C05477=1230.678,265.169,-62.603,-176.696,6.427,148.193
C05478=1230.673,265.417,-62.630,-176.693,6.429,148.193
C05479=1230.669,265.666,-62.657,-176.691,6.431,148.193
C05480=1230.665,265.914,-62.685,-176.689,6.433,148.193
C05481=1230.660,266.163,-62.713,-176.686,6.435,148.192
C05482=1230.656,266.411,-62.740,-176.684,6.437,148.192
C05483=1230.651,266.659,-62.767,-176.681,6.439,148.192
C05484=1230.647,266.908,-62.795,-176.679,6.441,148.192
C05485=1230.642,267.157,-62.822,-176.677,6.443,148.191
C05486=1230.638,267.405,-62.850,-176.674,6.445,148.191
C05487=1230.633,267.653,-62.877,-176.672,6.447,148.191
C05488=1230.629,267.903,-62.904,-176.669,6.449,148.191
C05489=1230.625,268.150,-62.932,-176.667,6.452,148.191
C05490=1230.620,268.399,-62.959,-176.664,6.454,148.190
C05491=1230.616,268.647,-62.987,-176.661,6.456,148.190
C05492=1230.612,268.896,-63.014,-176.659,6.458,148.190
C05493=1230.607,269.144,-63.041,-176.657,6.460,148.190
C05494=1230.603,269.392,-63.069,-176.655,6.462,148.190
C05495=1230.598,269.641,-63.096,-176.652,6.464,148.189
C05496=1230.595,269.889,-63.124,-176.649,6.466,148.189
C05497=1230.590,270.138,-63.151,-176.647,6.468,148.189
C05498=1230.585,270.386,-63.180,-176.645,6.470,148.189
C05499=1230.581,270.635,-63.207,-176.642,6.473,148.189
C05500=1230.576,270.883,-63.235,-176.639,6.475,148.188
C05501=1230.572,271.132,-63.262,-176.637,6.477,148.188
C05502=1230.568,271.380,-63.290,-176.635,6.479,148.188
C05503=1230.563,271.629,-63.317,-176.632,6.481,148.188
C05504=1230.559,271.877,-63.345,-176.630,6.483,148.188
C05505=1230.555,272.126,-63.374,-176.627,6.485,148.187
C05506=1230.550,272.374,-63.401,-176.625,6.487,148.187
C05507=1230.546,272.622,-63.428,-176.623,6.489,148.187
C05508=1230.541,272.871,-63.456,-176.620,6.492,148.187
C05509=1230.537,273.119,-63.484,-176.617,6.494,148.187
C05510=1230.533,273.367,-63.511,-176.615,6.496,148.187
C05511=1230.528,273.616,-63.539,-176.613,6.498,148.186
C05512=1230.524,273.864,-63.567,-176.610,6.500,148.186
C05513=1230.519,274.112,-63.595,-176.608,6.502,148.186
C05514=1230.515,274.361,-63.622,-176.605,6.504,148.186
C05515=1230.511,274.609,-63.650,-176.603,6.507,148.186
C05516=1230.506,274.858,-63.679,-176.600,6.509,148.185
C05517=1230.502,275.107,-63.706,-176.598,6.512,148.185
C05518=1230.497,275.354,-63.734,-176.595,6.513,148.185
C05519=1230.494,275.603,-63.762,-176.593,6.516,148.185
C05520=1230.489,275.851,-63.790,-176.591,6.518,148.185
C05521=1230.484,276.100,-63.818,-176.589,6.520,148.185
C05522=1230.480,276.348,-63.846,-176.586,6.522,148.184
C05523=1230.475,276.596,-63.874,-176.584,6.524,148.184
C05524=1230.471,276.845,-63.902,-176.581,6.527,148.184
C05525=1230.467,277.093,-63.929,-176.579,6.529,148.184
C05526=1230.463,277.342,-63.957,-176.576,6.531,148.184
C05527=1230.458,277.590,-63.986,-176.574,6.533,148.184
C05528=1230.454,277.839,-64.014,-176.571,6.535,148.183
C05529=1230.450,278.087,-64.042,-176.569,6.537,148.183
C05530=1230.445,278.335,-64.070,-176.567,6.539,148.183
C05531=1230.441,278.584,-64.097,-176.564,6.542,148.183
C05532=1230.436,278.832,-64.125,-176.561,6.544,148.183
C05533=1230.432,279.081,-64.154,-176.559,6.546,148.183
C05534=1230.427,279.329,-64.182,-176.557,6.548,148.182
C05535=1230.423,279.578,-64.210,-176.555,6.550,148.182
C05536=1230.419,279.825,-64.238,-176.552,6.552,148.182
C05537=1230.415,280.074,-64.266,-176.549,6.555,148.182
C05538=1230.410,280.322,-64.295,-176.547,6.557,148.182
C05539=1230.406,280.571,-64.323,-176.545,6.559,148.182
C05540=1230.401,280.819,-64.351,-176.543,6.562,148.181
C05541=1230.397,281.068,-64.379,-176.540,6.563,148.181
C05542=1230.393,281.315,-64.407,-176.538,6.566,148.181
C05543=1230.388,281.564,-64.436,-176.535,6.568,148.181
C05544=1230.384,281.812,-64.464,-176.533,6.571,148.181
C05545=1230.379,282.061,-64.492,-176.530,6.572,148.181
C05546=1230.375,282.309,-64.520,-176.528,6.575,148.180
C05547=1230.371,282.558,-64.549,-176.526,6.577,148.180
C05548=1230.366,282.806,-64.577,-176.523,6.579,148.180
C05549=1230.362,283.055,-64.605,-176.520,6.582,148.180
C05550=1230.357,283.303,-64.633,-176.518,6.584,148.180
C05551=1230.353,283.551,-64.662,-176.516,6.586,148.180
C05552=1230.349,283.799,-64.690,-176.513,6.588,148.179
C05553=1230.344,284.048,-64.718,-176.511,6.590,148.179
C05554=1230.340,284.297,-64.747,-176.509,6.592,148.179
C05555=1230.336,284.544,-64.776,-176.506,6.595,148.179
C05556=1230.332,284.793,-64.804,-176.504,6.597,148.179
C05557=1230.327,285.041,-64.832,-176.501,6.599,148.179
C05558=1230.323,285.290,-64.860,-176.499,6.601,148.179
C05559=1230.318,285.538,-64.889,-176.497,6.604,148.179
C05560=1230.314,285.786,-64.917,-176.494,6.606,148.178
C05561=1230.310,286.035,-64.946,-176.492,6.609,148.178
C05562=1230.305,286.283,-64.975,-176.490,6.611,148.178
C05563=1230.301,286.531,-65.003,-176.487,6.613,148.178
C05564=1230.296,286.780,-65.031,-176.485,6.615,148.178
C05565=1230.293,287.028,-65.060,-176.482,6.618,148.178
C05566=1230.288,287.276,-65.089,-176.480,6.620,148.178
C05567=1230.283,287.525,-65.117,-176.477,6.622,148.178
C05568=1230.279,287.773,-65.145,-176.475,6.624,148.177
C05569=1230.274,288.021,-65.174,-176.473,6.626,148.177
C05570=1230.271,288.269,-65.203,-176.470,6.629,148.177
C05571=1230.266,288.518,-65.231,-176.468,6.631,148.177
C05572=1230.261,288.766,-65.260,-176.465,6.633,148.177
C05573=1230.258,289.014,-65.288,-176.463,6.636,148.177
C05574=1230.253,289.289,-65.320,-176.460,6.638,148.177
C05575=1230.247,289.562,-65.351,-176.458,6.641,148.176
C05576=1230.243,289.836,-65.384,-176.455,6.643,148.176
C05577=1230.238,290.111,-65.415,-176.453,6.646,148.176
C05578=1230.234,290.359,-65.444,-176.450,6.647,148.176
C05579=1230.230,290.607,-65.473,-176.448,6.651,148.176
C05580=1230.225,290.856,-65.501,-176.445,6.653,148.176
C05581=1230.221,291.104,-65.530,-176.443,6.655,148.176
C05582=1230.216,291.352,-65.559,-176.441,6.657,148.175
C05583=1230.212,291.601,-65.587,-176.438,6.660,148.175
C05584=1230.208,291.849,-65.617,-176.436,6.662,148.175
C05585=1230.203,292.097,-65.645,-176.433,6.664,148.175
C05586=1230.199,292.345,-65.674,-176.431,6.666,148.175
C05587=1230.195,292.594,-65.703,-176.429,6.668,148.175
C05588=1230.191,292.842,-65.732,-176.426,6.671,148.175
C05589=1230.186,293.090,-65.761,-176.424,6.673,148.175
C05590=1230.181,293.339,-65.790,-176.422,6.676,148.175
C05591=1230.178,293.587,-65.818,-176.420,6.678,148.175
C05592=1230.173,293.835,-65.847,-176.417,6.681,148.174
C05593=1230.168,294.084,-65.876,-176.415,6.683,148.174
C05594=1230.164,294.332,-65.905,-176.412,6.685,148.174
C05595=1230.160,294.580,-65.935,-176.410,6.687,148.174
C05596=1230.156,294.828,-65.963,-176.408,6.689,148.174
C05597=1230.152,295.076,-65.992,-176.405,6.692,148.174
C05598=1230.147,295.325,-66.021,-176.403,6.694,148.174
C05599=1230.143,295.573,-66.050,-176.401,6.697,148.174
C05600=1230.138,295.821,-66.079,-176.398,6.699,148.173
C05601=1230.134,296.070,-66.108,-176.396,6.702,148.173
C05602=1230.130,296.318,-66.137,-176.393,6.704,148.173
C05603=1230.126,296.566,-66.166,-176.391,6.706,148.173
C05604=1230.122,296.815,-66.195,-176.389,6.708,148.173
C05605=1230.117,297.063,-66.224,-176.386,6.711,148.173
C05606=1230.113,297.311,-66.254,-176.384,6.713,148.173
C05607=1230.108,297.559,-66.283,-176.382,6.715,148.173
C05608=1230.104,297.808,-66.312,-176.380,6.718,148.173
C05609=1230.100,298.056,-66.341,-176.377,6.720,148.173
C05610=1230.095,298.304,-66.370,-176.375,6.723,148.173
C05611=1230.091,298.552,-66.400,-176.372,6.725,148.173
C05612=1230.086,298.801,-66.429,-176.370,6.727,148.172
C05613=1230.082,299.049,-66.458,-176.368,6.730,148.172
C05614=1230.079,299.297,-66.487,-176.365,6.732,148.172
C05615=1230.074,299.545,-66.516,-176.363,6.734,148.172
C05616=1230.070,299.793,-66.546,-176.361,6.737,148.172
C05617=1230.065,300.041,-66.575,-176.358,6.740,148.172
C05618=1230.061,300.290,-66.604,-176.356,6.742,148.172
C05619=1230.057,300.538,-66.633,-176.354,6.744,148.172
C05620=1230.053,300.787,-66.663,-176.351,6.746,148.172
C05621=1230.048,301.034,-66.692,-176.349,6.749,148.172
C05622=1230.044,301.283,-66.721,-176.347,6.751,148.172
C05623=1230.039,301.531,-66.751,-176.345,6.753,148.172
C05624=1230.035,301.779,-66.781,-176.342,6.756,148.172
C05625=1230.030,302.028,-66.810,-176.340,6.759,148.172
C05626=1230.026,302.276,-66.840,-176.338,6.761,148.171
C05627=1230.022,302.524,-66.869,-176.336,6.763,148.171
C05628=1230.018,302.773,-66.898,-176.333,6.765,148.171
C05629=1230.013,303.021,-66.927,-176.330,6.768,148.171
C05630=1230.009,303.269,-66.956,-176.328,6.770,148.171
C05631=1230.004,303.517,-66.986,-176.326,6.773,148.171
C05632=1230.000,303.765,-67.015,-176.324,6.775,148.171
C05633=1229.996,304.014,-67.045,-176.321,6.778,148.171
C05634=1229.992,304.262,-67.074,-176.319,6.780,148.171
C05635=1229.988,304.510,-67.104,-176.317,6.782,148.171
C05636=1229.983,304.758,-67.134,-176.315,6.785,148.171
C05637=1229.979,305.007,-67.164,-176.312,6.788,148.171
C05638=1229.975,305.255,-67.193,-176.310,6.789,148.171
C05639=1229.970,305.502,-67.222,-176.308,6.792,148.170
C05640=1229.966,305.751,-67.252,-176.306,6.794,148.170
C05641=1229.962,305.999,-67.281,-176.303,6.797,148.170
C05642=1229.957,306.247,-67.311,-176.301,6.799,148.170
C05643=1229.952,306.496,-67.341,-176.299,6.801,148.170
C05644=1229.948,306.744,-67.370,-176.296,6.805,148.170
C05645=1229.944,306.992,-67.400,-176.294,6.807,148.170
C05646=1229.940,307.240,-67.430,-176.292,6.809,148.170
C05647=1229.936,307.488,-67.459,-176.290,6.811,148.170
C05648=1229.931,307.737,-67.489,-176.287,6.814,148.170
C05649=1229.927,307.985,-67.519,-176.285,6.816,148.170
C05650=1229.923,308.233,-67.548,-176.283,6.819,148.170
C05651=1229.919,308.481,-67.578,-176.280,6.822,148.170
C05652=1229.914,308.730,-67.608,-176.278,6.824,148.170
C05653=1229.910,308.978,-67.638,-176.276,6.826,148.170
C05654=1229.906,309.226,-67.667,-176.274,6.828,148.170
C05655=1229.902,309.474,-67.698,-176.271,6.831,148.170
C05656=1229.897,309.722,-67.728,-176.269,6.834,148.170
C05657=1229.893,309.971,-67.757,-176.267,6.836,148.170
C05658=1229.889,310.218,-67.787,-176.265,6.838,148.170
C05659=1229.885,310.466,-67.817,-176.262,6.841,148.170
C05660=1229.880,310.715,-67.847,-176.260,6.843,148.170
C05661=1229.876,310.963,-67.877,-176.258,6.846,148.170
C05662=1229.872,311.211,-67.906,-176.256,6.849,148.170
C05663=1229.867,311.460,-67.936,-176.253,6.851,148.170
C05664=1229.863,311.707,-67.967,-176.251,6.853,148.169
C05665=1229.859,311.955,-67.996,-176.249,6.855,148.169
C05666=1229.854,312.204,-68.026,-176.247,6.858,148.169
C05667=1229.850,312.452,-68.056,-176.245,6.861,148.169
C05668=1229.846,312.700,-68.086,-176.242,6.863,148.169
C05669=1229.841,312.948,-68.116,-176.240,6.866,148.169
C05670=1229.837,313.196,-68.146,-176.238,6.868,148.170
C05671=1229.832,313.444,-68.177,-176.236,6.871,148.169
C05672=1229.828,313.692,-68.206,-176.234,6.873,148.169
C05673=1229.824,313.941,-68.236,-176.231,6.876,148.169
C05674=1229.820,314.189,-68.267,-176.229,6.878,148.169
C05675=1229.816,314.438,-68.296,-176.227,6.880,148.169
C05676=1229.811,314.686,-68.327,-176.224,6.883,148.169
C05677=1229.807,314.934,-68.356,-176.222,6.886,148.169
C05678=1229.803,315.209,-68.390,-176.220,6.889,148.169
C05679=1229.797,315.485,-68.423,-176.218,6.891,148.169
C05680=1229.793,315.760,-68.457,-176.215,6.894,148.169
C05681=1229.788,316.037,-68.490,-176.212,6.897,148.169
C05682=1229.784,316.285,-68.521,-176.211,6.900,148.169
C05683=1229.780,316.532,-68.551,-176.209,6.902,148.169
C05684=1229.775,316.781,-68.581,-176.206,6.904,148.169
C05685=1229.771,317.029,-68.612,-176.204,6.907,148.169
C05686=1229.767,317.277,-68.641,-176.202,6.909,148.169
C05687=1229.762,317.525,-68.672,-176.200,6.912,148.169
C05688=1229.759,317.773,-68.702,-176.197,6.915,148.169
C05689=1229.754,318.022,-68.732,-176.195,6.917,148.169
C05690=1229.750,318.270,-68.763,-176.193,6.919,148.169
C05691=1229.745,318.517,-68.793,-176.191,6.922,148.169
C05692=1229.741,318.766,-68.823,-176.188,6.925,148.169
C05693=1229.736,319.014,-68.854,-176.186,6.927,148.169
C05694=1229.733,319.262,-68.884,-176.185,6.929,148.169
C05695=1229.728,319.511,-68.914,-176.182,6.933,148.169
C05696=1229.724,319.759,-68.945,-176.180,6.935,148.169
C05697=1229.720,320.006,-68.975,-176.178,6.937,148.169
C05698=1229.715,320.254,-69.006,-176.175,6.940,148.169
C05699=1229.712,320.503,-69.036,-176.174,6.943,148.170
C05700=1229.707,320.751,-69.066,-176.172,6.945,148.169
C05701=1229.703,320.999,-69.097,-176.169,6.947,148.169
C05702=1229.698,321.247,-69.127,-176.167,6.950,148.169
C05703=1229.694,321.495,-69.158,-176.165,6.953,148.170
C05704=1229.690,321.744,-69.188,-176.163,6.955,148.170
C05705=1229.686,321.992,-69.219,-176.160,6.958,148.170
C05706=1229.681,322.240,-69.249,-176.158,6.960,148.170
C05707=1229.677,322.487,-69.280,-176.157,6.963,148.170
C05708=1229.673,322.735,-69.310,-176.155,6.965,148.170
C05709=1229.669,322.984,-69.341,-176.152,6.968,148.170
C05710=1229.665,323.231,-69.372,-176.150,6.970,148.170
C05711=1229.660,323.479,-69.402,-176.148,6.973,148.170
C05712=1229.656,323.728,-69.432,-176.146,6.976,148.170
C05713=1229.652,323.976,-69.463,-176.144,6.978,148.170
C05714=1229.647,324.224,-69.494,-176.142,6.981,148.170
C05715=1229.643,324.472,-69.524,-176.139,6.984,148.170
C05716=1229.639,324.720,-69.555,-176.137,6.986,148.170
C05717=1229.635,324.969,-69.586,-176.135,6.988,148.170
C05718=1229.630,325.217,-69.617,-176.133,6.991,148.170
C05719=1229.626,325.464,-69.647,-176.131,6.994,148.170
C05720=1229.622,325.713,-69.678,-176.129,6.996,148.170
C05721=1229.618,325.961,-69.709,-176.127,6.998,148.170
C05722=1229.614,326.208,-69.739,-176.125,7.002,148.170
C05723=1229.610,326.457,-69.770,-176.123,7.004,148.170
C05724=1229.605,326.705,-69.801,-176.121,7.006,148.170
C05725=1229.601,326.953,-69.832,-176.119,7.009,148.170
C05726=1229.596,327.201,-69.862,-176.116,7.012,148.170
C05727=1229.593,327.449,-69.894,-176.114,7.014,148.170
C05728=1229.588,327.697,-69.924,-176.113,7.017,148.171
C05729=1229.584,327.945,-69.955,-176.110,7.020,148.171
C05730=1229.580,328.193,-69.986,-176.108,7.022,148.171
C05731=1229.575,328.441,-70.017,-176.106,7.024,148.171
C05732=1229.571,328.689,-70.047,-176.104,7.027,148.171
C05733=1229.567,328.938,-70.078,-176.102,7.030,148.171
C05734=1229.563,329.185,-70.109,-176.100,7.032,148.171
C05735=1229.558,329.433,-70.140,-176.098,7.035,148.171
C05736=1229.554,329.681,-70.172,-176.096,7.038,148.171
C05737=1229.550,329.929,-70.202,-176.094,7.040,148.171
C05738=1229.546,330.177,-70.233,-176.092,7.043,148.171
C05739=1229.542,330.426,-70.264,-176.090,7.046,148.171
C05740=1229.537,330.674,-70.294,-176.088,7.048,148.171
C05741=1229.533,330.922,-70.326,-176.086,7.050,148.171
C05742=1229.529,331.170,-70.357,-176.084,7.053,148.172
C05743=1229.524,331.418,-70.388,-176.081,7.056,148.172
C05744=1229.520,331.666,-70.419,-176.080,7.059,148.172
C05745=1229.516,331.914,-70.450,-176.078,7.061,148.172
C05746=1229.511,332.162,-70.481,-176.075,7.064,148.172
C05747=1229.508,332.410,-70.512,-176.073,7.066,148.172
C05748=1229.504,332.657,-70.543,-176.072,7.069,148.172
C05749=1229.500,332.906,-70.574,-176.070,7.071,148.172
C05750=1229.495,333.154,-70.605,-176.067,7.074,148.172
C05751=1229.491,333.401,-70.637,-176.066,7.077,148.172
C05752=1229.487,333.650,-70.668,-176.064,7.079,148.172
C05753=1229.482,333.898,-70.698,-176.061,7.083,148.173
C05754=1229.478,334.146,-70.730,-176.059,7.085,148.173
C05755=1229.474,334.394,-70.761,-176.058,7.087,148.173
C05756=1229.470,334.643,-70.792,-176.056,7.090,148.173
C05757=1229.466,334.890,-70.824,-176.053,7.093,148.173
C05758=1229.461,335.138,-70.854,-176.051,7.095,148.173
C05759=1229.457,335.386,-70.886,-176.050,7.098,148.173
C05760=1229.453,335.634,-70.917,-176.048,7.101,148.173
C05761=1229.449,335.882,-70.949,-176.045,7.103,148.173
C05762=1229.444,336.130,-70.980,-176.044,7.106,148.173
C05763=1229.441,336.378,-71.012,-176.042,7.108,148.173
C05764=1229.436,336.626,-71.042,-176.040,7.111,148.174
C05765=1229.432,336.874,-71.074,-176.038,7.114,148.174
C05766=1229.428,337.122,-71.105,-176.036,7.116,148.174
C05767=1229.424,337.370,-71.137,-176.034,7.120,148.174
C05768=1229.419,337.618,-71.168,-176.032,7.122,148.174
C05769=1229.415,337.866,-71.200,-176.030,7.124,148.174
C05770=1229.410,338.114,-71.231,-176.028,7.127,148.174
C05771=1229.406,338.361,-71.262,-176.026,7.130,148.175
C05772=1229.402,338.610,-71.293,-176.024,7.132,148.175
C05773=1229.398,338.858,-71.325,-176.022,7.135,148.175
C05774=1229.394,339.106,-71.356,-176.021,7.138,148.175
C05775=1229.390,339.354,-71.388,-176.018,7.141,148.175
C05776=1229.386,339.601,-71.419,-176.017,7.143,148.175
C05777=1229.382,339.850,-71.450,-176.015,7.146,148.175
C05778=1229.377,340.097,-71.482,-176.013,7.148,148.175
C05779=1229.373,340.346,-71.514,-176.011,7.151,148.175
C05780=1229.368,340.594,-71.545,-176.009,7.154,148.176
C05781=1229.365,340.842,-71.577,-176.007,7.156,148.176
C05782=1229.359,341.119,-71.611,-176.005,7.159,148.176
C05783=1229.355,341.397,-71.647,-176.003,7.163,148.176
C05784=1229.351,341.674,-71.683,-176.001,7.165,148.176
C05785=1229.345,341.953,-71.718,-175.998,7.168,148.176
C05786=1229.341,342.200,-71.750,-175.997,7.171,148.176
C05787=1229.337,342.448,-71.781,-175.995,7.173,148.177
C05788=1229.333,342.696,-71.813,-175.993,7.177,148.177
C05789=1229.329,342.944,-71.844,-175.991,7.179,148.177
C05790=1229.324,343.192,-71.876,-175.989,7.182,148.177
C05791=1229.320,343.440,-71.908,-175.988,7.184,148.177
C05792=1229.316,343.687,-71.939,-175.985,7.187,148.177
C05793=1229.312,343.936,-71.971,-175.984,7.190,148.178
C05794=1229.307,344.184,-72.003,-175.982,7.192,148.178
C05795=1229.303,344.432,-72.035,-175.980,7.195,148.178
C05796=1229.299,344.680,-72.066,-175.978,7.198,148.178
C05797=1229.295,344.927,-72.098,-175.976,7.201,148.178
C05798=1229.291,345.175,-72.130,-175.975,7.203,148.178
C05799=1229.287,345.424,-72.161,-175.973,7.206,148.179
C05800=1229.282,345.671,-72.193,-175.971,7.209,148.179
C05801=1229.278,345.920,-72.225,-175.969,7.211,148.179
C05802=1229.274,346.167,-72.257,-175.967,7.214,148.179
C05803=1229.270,346.415,-72.289,-175.965,7.216,148.179
C05804=1229.265,346.663,-72.321,-175.963,7.220,148.179
C05805=1229.261,346.911,-72.353,-175.962,7.222,148.180
C05806=1229.257,347.159,-72.384,-175.960,7.225,148.180
C05807=1229.253,347.407,-72.417,-175.958,7.227,148.180
C05808=1229.249,347.654,-72.448,-175.957,7.230,148.180
C05809=1229.245,347.903,-72.479,-175.955,7.233,148.180
C05810=1229.240,348.151,-72.512,-175.953,7.236,148.180
C05811=1229.236,348.399,-72.543,-175.951,7.238,148.181
C05812=1229.232,348.647,-72.575,-175.949,7.240,148.181
C05813=1229.227,348.894,-72.607,-175.947,7.244,148.181
C05814=1229.223,349.142,-72.639,-175.946,7.246,148.181
C05815=1229.219,349.391,-72.672,-175.944,7.249,148.181
C05816=1229.215,349.638,-72.703,-175.942,7.251,148.181
C05817=1229.211,349.886,-72.736,-175.941,7.254,148.182
C05818=1229.207,350.134,-72.768,-175.938,7.257,148.182
C05819=1229.203,350.381,-72.800,-175.937,7.260,148.182
C05820=1229.198,350.630,-72.832,-175.935,7.262,148.182
C05821=1229.194,350.878,-72.864,-175.934,7.265,148.182
C05822=1229.191,351.126,-72.896,-175.932,7.267,148.183
C05823=1229.186,351.373,-72.928,-175.930,7.271,148.183
C05824=1229.182,351.621,-72.960,-175.928,7.273,148.183
C05825=1229.178,351.870,-72.992,-175.927,7.276,148.183
C05826=1229.173,352.117,-73.024,-175.925,7.278,148.183
C05827=1229.169,352.365,-73.057,-175.924,7.281,148.184
C05828=1229.165,352.613,-73.089,-175.922,7.285,148.184
C05829=1229.160,352.860,-73.121,-175.920,7.287,148.184
C05830=1229.157,353.109,-73.152,-175.918,7.290,148.184
C05831=1229.152,353.357,-73.185,-175.917,7.292,148.185
C05832=1229.148,353.605,-73.217,-175.915,7.295,148.185
C05833=1229.144,353.852,-73.250,-175.913,7.298,148.185
C05834=1229.140,354.100,-73.281,-175.911,7.301,148.185
C05835=1229.136,354.348,-73.314,-175.910,7.303,148.185
C05836=1229.132,354.596,-73.346,-175.908,7.306,148.185
C05837=1229.127,354.843,-73.378,-175.907,7.309,148.186
C05838=1229.123,355.091,-73.410,-175.905,7.312,148.186
C05839=1229.119,355.340,-73.443,-175.903,7.314,148.186
C05840=1229.115,355.588,-73.475,-175.901,7.317,148.187
C05841=1229.111,355.835,-73.507,-175.900,7.319,148.187
C05842=1229.106,356.083,-73.540,-175.898,7.322,148.187
C05843=1229.102,356.331,-73.572,-175.897,7.325,148.187
C05844=1229.098,356.579,-73.605,-175.895,7.328,148.188
C05845=1229.095,356.827,-73.637,-175.893,7.331,148.188
C05846=1229.089,357.075,-73.669,-175.892,7.333,148.188
C05847=1229.086,357.322,-73.701,-175.890,7.336,148.188
C05848=1229.082,357.570,-73.734,-175.888,7.338,148.188
C05849=1229.077,357.819,-73.766,-175.887,7.341,148.189
C05850=1229.074,358.066,-73.799,-175.886,7.344,148.189
C05851=1229.069,358.314,-73.831,-175.883,7.347,148.189
C05852=1229.065,358.562,-73.863,-175.882,7.350,148.189
C05853=1229.061,358.810,-73.896,-175.881,7.352,148.190
C05854=1229.056,359.058,-73.928,-175.879,7.355,148.190
C05855=1229.053,359.305,-73.961,-175.877,7.357,148.190
C05856=1229.048,359.553,-73.993,-175.876,7.360,148.190
C05857=1229.044,359.801,-74.026,-175.875,7.363,148.191
C05858=1229.040,360.049,-74.058,-175.872,7.366,148.191
C05859=1229.036,360.297,-74.090,-175.871,7.369,148.191
C05860=1229.032,360.545,-74.123,-175.870,7.372,148.191
C05861=1229.028,360.793,-74.155,-175.868,7.374,148.192
C05862=1229.023,361.040,-74.188,-175.866,7.377,148.192
C05863=1229.019,361.288,-74.221,-175.865,7.379,148.192
C05864=1229.015,361.536,-74.253,-175.864,7.382,148.192
C05865=1229.011,361.784,-74.286,-175.862,7.384,148.193
C05866=1229.007,362.032,-74.319,-175.861,7.387,148.193
C05867=1229.003,362.280,-74.352,-175.859,7.391,148.193
C05868=1228.999,362.528,-74.384,-175.857,7.393,148.193
C05869=1228.994,362.775,-74.417,-175.856,7.396,148.194
C05870=1228.990,363.023,-74.449,-175.854,7.399,148.194
C05871=1228.986,363.271,-74.482,-175.853,7.401,148.194
C05872=1228.982,363.519,-74.514,-175.851,7.404,148.195
C05873=1228.978,363.766,-74.547,-175.850,7.406,148.195
C05874=1228.974,364.014,-74.580,-175.849,7.409,148.195
C05875=1228.969,364.263,-74.613,-175.847,7.412,148.195
C05876=1228.966,364.510,-74.645,-175.846,7.415,148.196
C05877=1228.962,364.758,-74.678,-175.844,7.417,148.196
C05878=1228.957,365.006,-74.711,-175.843,7.420,148.196
C05879=1228.952,365.253,-74.744,-175.841,7.423,148.197
C05880=1228.949,365.501,-74.775,-175.840,7.426,148.197
C05881=1228.945,365.749,-74.809,-175.838,7.429,148.197
C05882=1228.940,365.997,-74.842,-175.837,7.432,148.198
C05883=1228.936,366.244,-74.875,-175.835,7.434,148.198
C05884=1228.932,366.493,-74.907,-175.834,7.437,148.198
C05885=1228.928,366.740,-74.940,-175.832,7.439,148.198
C05886=1228.924,367.020,-74.977,-175.831,7.442,148.199
C05887=1228.919,367.300,-75.014,-175.829,7.446,148.199
C05888=1228.914,367.579,-75.051,-175.828,7.448,148.199
C05889=1228.910,367.858,-75.088,-175.826,7.452,148.200
C05890=1228.905,368.106,-75.121,-175.825,7.455,148.200
C05891=1228.901,368.354,-75.154,-175.823,7.457,148.200
C05892=1228.897,368.602,-75.187,-175.822,7.460,148.201
C05893=1228.893,368.850,-75.220,-175.821,7.463,148.201
C05894=1228.889,369.097,-75.253,-175.819,7.465,148.201
C05895=1228.884,369.346,-75.286,-175.818,7.468,148.202
C05896=1228.880,369.593,-75.319,-175.816,7.471,148.202
C05897=1228.876,369.841,-75.352,-175.815,7.474,148.202
C05898=1228.873,370.088,-75.385,-175.814,7.476,148.203
C05899=1228.869,370.336,-75.418,-175.813,7.478,148.203
C05900=1228.864,370.584,-75.451,-175.812,7.481,148.203
C05901=1228.860,370.832,-75.484,-175.811,7.484,148.203
C05902=1228.856,371.080,-75.517,-175.809,7.486,148.204
C05903=1228.852,371.328,-75.550,-175.808,7.489,148.204
C05904=1228.848,371.575,-75.583,-175.807,7.492,148.204
C05905=1228.843,371.823,-75.616,-175.805,7.494,148.205
C05906=1228.839,372.071,-75.649,-175.804,7.497,148.205
C05907=1228.835,372.319,-75.682,-175.803,7.500,148.205
C05908=1228.831,372.566,-75.716,-175.801,7.503,148.206
C05909=1228.827,372.814,-75.749,-175.800,7.505,148.206
C05910=1228.823,373.062,-75.782,-175.799,7.508,148.206
C05911=1228.818,373.310,-75.814,-175.798,7.511,148.207
C05912=1228.814,373.558,-75.848,-175.796,7.514,148.207
C05913=1228.810,373.806,-75.881,-175.795,7.516,148.207
C05914=1228.806,374.053,-75.914,-175.794,7.519,148.208
C05915=1228.802,374.301,-75.947,-175.792,7.522,148.208
C05916=1228.798,374.549,-75.980,-175.791,7.524,148.208
C05917=1228.794,374.797,-76.013,-175.790,7.527,148.209
C05918=1228.789,375.044,-76.046,-175.789,7.529,148.209
C05919=1228.785,375.292,-76.080,-175.788,7.532,148.210
C05920=1228.781,375.540,-76.113,-175.786,7.535,148.210
C05921=1228.777,375.787,-76.146,-175.785,7.538,148.210
C05922=1228.773,376.035,-76.180,-175.784,7.540,148.211
C05923=1228.769,376.282,-76.213,-175.783,7.543,148.211
C05924=1228.765,376.530,-76.246,-175.782,7.545,148.211
C05925=1228.761,376.778,-76.279,-175.780,7.548,148.211
C05926=1228.757,377.025,-76.312,-175.779,7.551,148.212
C05927=1228.752,377.273,-76.346,-175.778,7.553,148.212
C05928=1228.748,377.521,-76.379,-175.777,7.556,148.213
C05929=1228.744,377.769,-76.412,-175.776,7.559,148.213
C05930=1228.741,378.017,-76.445,-175.775,7.561,148.213
C05931=1228.737,378.265,-76.479,-175.774,7.564,148.214
C05932=1228.732,378.513,-76.512,-175.772,7.566,148.214
C05933=1228.728,378.760,-76.546,-175.771,7.569,148.214
C05934=1228.724,379.008,-76.579,-175.770,7.572,148.215
C05935=1228.720,379.255,-76.613,-175.769,7.575,148.215
C05936=1228.715,379.503,-76.646,-175.768,7.577,148.216
C05937=1228.711,379.751,-76.679,-175.767,7.580,148.216
C05938=1228.707,379.999,-76.712,-175.766,7.582,148.216
C05939=1228.703,380.246,-76.746,-175.765,7.585,148.217
C05940=1228.698,380.494,-76.780,-175.764,7.587,148.217
C05941=1228.695,380.742,-76.813,-175.762,7.590,148.217
C05942=1228.691,380.990,-76.846,-175.761,7.593,148.218
C05943=1228.687,381.238,-76.879,-175.760,7.595,148.218
C05944=1228.683,381.485,-76.913,-175.759,7.598,148.218
C05945=1228.679,381.733,-76.946,-175.758,7.600,148.219
C05946=1228.674,381.980,-76.980,-175.757,7.603,148.219
C05947=1228.670,382.228,-77.013,-175.756,7.606,148.220
C05948=1228.666,382.475,-77.047,-175.755,7.609,148.220
C05949=1228.662,382.724,-77.081,-175.754,7.611,148.220
C05950=1228.658,382.972,-77.114,-175.753,7.614,148.221
C05951=1228.654,383.219,-77.147,-175.752,7.616,148.221
C05952=1228.649,383.467,-77.182,-175.751,7.618,148.221
C05953=1228.645,383.714,-77.215,-175.750,7.621,148.222
C05954=1228.641,383.962,-77.248,-175.749,7.624,148.222
C05955=1228.637,384.209,-77.282,-175.748,7.627,148.223
C05956=1228.634,384.458,-77.315,-175.747,7.629,148.223
C05957=1228.629,384.706,-77.349,-175.746,7.632,148.223
C05958=1228.625,384.953,-77.383,-175.745,7.634,148.224
C05959=1228.621,385.201,-77.416,-175.744,7.636,148.224
C05960=1228.617,385.448,-77.449,-175.743,7.639,148.225
C05961=1228.612,385.696,-77.484,-175.742,7.642,148.225
C05962=1228.608,385.943,-77.517,-175.741,7.644,148.225
C05963=1228.605,386.192,-77.550,-175.740,7.647,148.226
C05964=1228.601,386.439,-77.584,-175.739,7.650,148.226
C05965=1228.596,386.687,-77.618,-175.738,7.652,148.226
C05966=1228.592,386.934,-77.652,-175.738,7.655,148.227
C05967=1228.588,387.182,-77.685,-175.736,7.658,148.227
C05968=1228.584,387.430,-77.718,-175.736,7.660,148.228
C05969=1228.580,387.678,-77.753,-175.735,7.662,148.228
C05970=1228.576,387.925,-77.786,-175.733,7.665,148.229
C05971=1228.572,388.173,-77.820,-175.733,7.667,148.229
C05972=1228.567,388.421,-77.854,-175.732,7.670,148.229
C05973=1228.564,388.668,-77.888,-175.731,7.672,148.230
C05974=1228.560,388.916,-77.921,-175.730,7.675,148.230
C05975=1228.556,389.163,-77.955,-175.729,7.678,148.230
C05976=1228.551,389.411,-77.989,-175.728,7.680,148.231
C05977=1228.547,389.658,-78.023,-175.727,7.683,148.231
C05978=1228.543,389.907,-78.056,-175.727,7.685,148.232
C05979=1228.539,390.154,-78.091,-175.725,7.688,148.232
C05980=1228.535,390.402,-78.124,-175.724,7.690,148.233
C05981=1228.531,390.649,-78.158,-175.724,7.692,148.233
C05982=1228.526,390.897,-78.191,-175.723,7.695,148.233
C05983=1228.523,391.145,-78.226,-175.722,7.697,148.234
C05984=1228.519,391.393,-78.259,-175.721,7.700,148.234
C05985=1228.514,391.640,-78.293,-175.721,7.702,148.235
C05986=1228.510,391.888,-78.326,-175.719,7.705,148.235
C05987=1228.506,392.136,-78.361,-175.718,7.708,148.235
C05988=1228.502,392.384,-78.394,-175.718,7.710,148.236
C05989=1228.498,392.631,-78.428,-175.716,7.713,148.236
C05990=1228.494,392.913,-78.466,-175.716,7.715,148.237
C05991=1228.488,393.194,-78.505,-175.715,7.718,148.237
C05992=1228.484,393.475,-78.544,-175.714,7.721,148.237
C05993=1228.479,393.757,-78.582,-175.713,7.724,148.238
C05994=1228.476,394.004,-78.616,-175.712,7.727,148.239
C05995=1228.471,394.252,-78.650,-175.711,7.729,148.239
C05996=1228.467,394.499,-78.684,-175.710,7.731,148.239
C05997=1228.463,394.747,-78.719,-175.710,7.733,148.240
C05998=1228.459,394.995,-78.752,-175.709,7.736,148.240
C05999=1228.455,395.242,-78.786,-175.708,7.738,148.241
C06000=1228.451,395.490,-78.821,-175.708,7.740,148.241
C06001=1228.447,395.738,-78.854,-175.706,7.743,148.241
C06002=1228.442,395.985,-78.888,-175.706,7.745,148.242
C06003=1228.439,396.232,-78.922,-175.705,7.748,148.242
C06004=1228.434,396.481,-78.956,-175.704,7.750,148.243
C06005=1228.430,396.728,-78.990,-175.703,7.753,148.243
C06006=1228.426,396.976,-79.025,-175.703,7.755,148.243
C06007=1228.422,397.224,-79.058,-175.702,7.758,148.244
C06008=1228.418,397.471,-79.092,-175.701,7.760,148.244
C06009=1228.414,397.719,-79.126,-175.701,7.762,148.245
C06010=1228.410,397.966,-79.160,-175.700,7.765,148.245
C06011=1228.406,398.215,-79.194,-175.699,7.767,148.245
C06012=1228.402,398.462,-79.228,-175.698,7.770,148.246
C06013=1228.397,398.709,-79.263,-175.698,7.772,148.246
C06014=1228.394,398.958,-79.296,-175.696,7.775,148.247
C06015=1228.389,399.205,-79.331,-175.696,7.777,148.247
C06016=1228.385,399.452,-79.365,-175.696,7.779,148.248
C06017=1228.381,399.700,-79.399,-175.694,7.782,148.248
C06018=1228.377,399.948,-79.433,-175.694,7.784,148.248
C06019=1228.373,400.195,-79.467,-175.693,7.786,148.249
C06020=1228.370,400.443,-79.501,-175.692,7.789,148.249
C06021=1228.365,400.691,-79.536,-175.692,7.791,148.250
C06022=1228.361,400.938,-79.570,-175.691,7.794,148.250
C06023=1228.357,401.186,-79.604,-175.690,7.796,148.250
C06024=1228.353,401.434,-79.638,-175.690,7.798,148.251
C06025=1228.348,401.681,-79.672,-175.689,7.801,148.251
C06026=1228.345,401.929,-79.706,-175.688,7.803,148.252
C06027=1228.341,402.176,-79.741,-175.687,7.805,148.252
C06028=1228.336,402.424,-79.775,-175.687,7.808,148.253
C06029=1228.333,402.672,-79.809,-175.686,7.810,148.253
C06030=1228.328,402.919,-79.843,-175.685,7.812,148.253
C06031=1228.324,403.167,-79.877,-175.685,7.815,148.254
C06032=1228.320,403.415,-79.912,-175.684,7.817,148.254
C06033=1228.316,403.662,-79.946,-175.683,7.819,148.255
C06034=1228.312,403.909,-79.980,-175.682,7.822,148.255
C06035=1228.309,404.157,-80.015,-175.682,7.824,148.255
C06036=1228.304,404.405,-80.048,-175.681,7.826,148.256
C06037=1228.299,404.652,-80.083,-175.681,7.828,148.256
C06038=1228.296,404.900,-80.117,-175.680,7.831,148.257
C06039=1228.291,405.148,-80.152,-175.679,7.833,148.257
C06040=1228.287,405.395,-80.185,-175.679,7.835,148.257
C06041=1228.284,405.643,-80.220,-175.678,7.838,148.258
C06042=1228.279,405.890,-80.255,-175.678,7.840,148.258
C06043=1228.276,406.138,-80.289,-175.677,7.842,148.259
C06044=1228.271,406.386,-80.323,-175.676,7.844,148.259
C06045=1228.267,406.633,-80.357,-175.675,7.847,148.259
C06046=1228.263,406.881,-80.392,-175.675,7.849,148.260
C06047=1228.259,407.128,-80.427,-175.674,7.851,148.260
C06048=1228.256,407.376,-80.461,-175.674,7.853,148.261
C06049=1228.251,407.623,-80.495,-175.673,7.856,148.261
C06050=1228.247,407.871,-80.529,-175.672,7.858,148.262
C06051=1228.243,408.119,-80.564,-175.672,7.860,148.262
C06052=1228.239,408.366,-80.598,-175.671,7.862,148.262
C06053=1228.235,408.614,-80.633,-175.670,7.865,148.263
C06054=1228.231,408.861,-80.667,-175.670,7.867,148.263
C06055=1228.226,409.109,-80.702,-175.669,7.869,148.264
C06056=1228.223,409.357,-80.736,-175.669,7.872,148.264
C06057=1228.218,409.604,-80.770,-175.668,7.874,148.265
C06058=1228.214,409.852,-80.805,-175.667,7.877,148.265
C06059=1228.211,410.099,-80.839,-175.666,7.878,148.265
C06060=1228.206,410.347,-80.873,-175.666,7.881,148.266
C06061=1228.202,410.595,-80.908,-175.666,7.883,148.266
C06062=1228.198,410.842,-80.942,-175.665,7.885,148.266
C06063=1228.194,411.090,-80.977,-175.664,7.888,148.267
C06064=1228.190,411.337,-81.011,-175.664,7.890,148.267
C06065=1228.186,411.585,-81.045,-175.663,7.892,148.268
C06066=1228.182,411.833,-81.080,-175.662,7.894,148.268
C06067=1228.177,412.080,-81.115,-175.662,7.896,148.269
C06068=1228.174,412.328,-81.149,-175.662,7.898,148.269
C06069=1228.170,412.575,-81.183,-175.660,7.901,148.269
C06070=1228.166,412.823,-81.218,-175.660,7.903,148.270
C06071=1228.162,413.070,-81.253,-175.660,7.905,148.270
C06072=1228.158,413.318,-81.288,-175.659,7.907,148.271
C06073=1228.154,413.565,-81.322,-175.658,7.909,148.271
C06074=1228.149,413.813,-81.357,-175.658,7.911,148.272
C06075=1228.146,414.061,-81.391,-175.657,7.913,148.272
C06076=1228.141,414.308,-81.425,-175.656,7.916,148.272
C06077=1228.137,414.556,-81.460,-175.656,7.918,148.273
C06078=1228.133,414.804,-81.495,-175.655,7.920,148.273
C06079=1228.130,415.051,-81.529,-175.655,7.922,148.273
C06080=1228.125,415.298,-81.564,-175.654,7.924,148.274
C06081=1228.121,415.546,-81.599,-175.654,7.927,148.274
C06082=1228.115,415.933,-81.653,-175.653,7.931,148.275
C06083=1228.109,416.320,-81.707,-175.652,7.934,148.276
C06084=1228.102,416.707,-81.761,-175.651,7.937,148.276
C06085=1228.097,417.094,-81.815,-175.651,7.940,148.277
C06086=1227.675,417.093,-81.847,-175.654,7.950,148.280
C06087=1227.680,416.704,-81.793,-175.654,7.947,148.280
C06088=1227.687,416.315,-81.739,-175.655,7.944,148.279
C06089=1227.693,415.925,-81.684,-175.656,7.940,148.279
C06090=1227.699,415.536,-81.630,-175.657,7.937,148.278
C06091=1227.703,415.288,-81.595,-175.658,7.935,148.278
C06092=1227.707,415.041,-81.561,-175.658,7.933,148.277
C06093=1227.711,414.792,-81.526,-175.659,7.931,148.277
C06094=1227.716,414.545,-81.492,-175.659,7.929,148.276
C06095=1227.720,414.298,-81.457,-175.660,7.926,148.276
C06096=1227.723,414.050,-81.422,-175.661,7.924,148.275
C06097=1227.728,413.803,-81.388,-175.661,7.922,148.275
C06098=1227.732,413.555,-81.353,-175.662,7.920,148.275
C06099=1227.735,413.308,-81.319,-175.662,7.918,148.274
C06100=1227.739,413.060,-81.284,-175.663,7.915,148.274
C06101=1227.744,412.812,-81.250,-175.663,7.913,148.274
C06102=1227.748,412.564,-81.215,-175.664,7.911,148.273
C06103=1227.751,412.318,-81.180,-175.665,7.908,148.273
C06104=1227.756,412.070,-81.146,-175.665,7.906,148.272
C06105=1227.760,411.822,-81.111,-175.666,7.904,148.272
C06106=1227.764,411.575,-81.077,-175.666,7.902,148.272
C06107=1227.768,411.327,-81.042,-175.667,7.900,148.271
C06108=1227.772,411.079,-81.008,-175.668,7.897,148.271
C06109=1227.776,410.832,-80.974,-175.668,7.895,148.270
C06110=1227.780,410.584,-80.939,-175.669,7.893,148.270
C06111=1227.785,410.337,-80.905,-175.669,7.891,148.269
C06112=1227.788,410.089,-80.871,-175.670,7.889,148.269
C06113=1227.792,409.842,-80.836,-175.670,7.887,148.269
C06114=1227.796,409.593,-80.801,-175.671,7.884,148.268
C06115=1227.800,409.346,-80.767,-175.672,7.882,148.268
C06116=1227.804,409.098,-80.733,-175.673,7.880,148.267
C06117=1227.809,408.851,-80.698,-175.673,7.878,148.267
C06118=1227.813,408.604,-80.664,-175.674,7.875,148.266
C06119=1227.817,408.356,-80.629,-175.675,7.873,148.266
C06120=1227.821,408.108,-80.595,-175.675,7.871,148.266
C06121=1227.824,407.860,-80.561,-175.675,7.869,148.265
C06122=1227.829,407.613,-80.526,-175.676,7.867,148.265
C06123=1227.834,407.365,-80.492,-175.677,7.864,148.264
C06124=1227.837,407.118,-80.458,-175.677,7.862,148.264
C06125=1227.841,406.870,-80.423,-175.678,7.860,148.264
C06126=1227.845,406.622,-80.389,-175.679,7.858,148.263
C06127=1227.849,406.375,-80.354,-175.679,7.855,148.263
C06128=1227.854,406.128,-80.320,-175.680,7.853,148.262
C06129=1227.857,405.880,-80.286,-175.681,7.851,148.262
C06130=1227.862,405.632,-80.251,-175.681,7.848,148.261
C06131=1227.865,405.385,-80.217,-175.682,7.846,148.261
C06132=1227.869,405.137,-80.182,-175.683,7.844,148.261
C06133=1227.874,404.890,-80.148,-175.683,7.842,148.260
C06134=1227.877,404.642,-80.114,-175.684,7.838,148.260
C06135=1227.882,404.394,-80.079,-175.685,7.836,148.259
C06136=1227.886,404.147,-80.045,-175.685,7.835,148.259
C06137=1227.890,403.899,-80.011,-175.685,7.832,148.259
C06138=1227.894,403.651,-79.977,-175.687,7.829,148.258
C06139=1227.898,403.404,-79.943,-175.687,7.827,148.258
C06140=1227.902,403.156,-79.908,-175.688,7.825,148.257
C06141=1227.906,402.909,-79.874,-175.689,7.822,148.257
C06142=1227.911,402.661,-79.840,-175.689,7.820,148.257
C06143=1227.914,402.414,-79.806,-175.690,7.818,148.256
C06144=1227.918,402.166,-79.771,-175.690,7.815,148.256
C06145=1227.923,401.918,-79.738,-175.691,7.813,148.255
C06146=1227.926,401.670,-79.703,-175.692,7.811,148.255
C06147=1227.931,401.423,-79.669,-175.693,7.808,148.254
C06148=1227.935,401.176,-79.635,-175.693,7.806,148.254
C06149=1227.939,400.928,-79.600,-175.694,7.804,148.254
C06150=1227.943,400.680,-79.567,-175.695,7.801,148.253
C06151=1227.948,400.433,-79.532,-175.696,7.799,148.253
C06152=1227.951,400.185,-79.498,-175.696,7.796,148.252
C06153=1227.955,399.937,-79.464,-175.697,7.794,148.252
C06154=1227.959,399.690,-79.430,-175.698,7.792,148.252
C06155=1227.963,399.441,-79.396,-175.699,7.790,148.251
C06156=1227.967,399.194,-79.362,-175.699,7.787,148.251
C06157=1227.972,398.947,-79.327,-175.700,7.784,148.250
C06158=1227.975,398.699,-79.293,-175.701,7.782,148.250
C06159=1227.980,398.451,-79.259,-175.701,7.780,148.250
C06160=1227.984,398.204,-79.225,-175.702,7.777,148.249
C06161=1227.988,397.956,-79.191,-175.703,7.775,148.249
C06162=1227.992,397.709,-79.157,-175.704,7.773,148.248
C06163=1227.996,397.461,-79.123,-175.704,7.771,148.248
C06164=1228.000,397.214,-79.089,-175.705,7.768,148.247
C06165=1228.004,396.965,-79.054,-175.706,7.765,148.247
C06166=1228.008,396.718,-79.020,-175.706,7.764,148.247
C06167=1228.012,396.471,-78.987,-175.708,7.761,148.246
C06168=1228.016,396.223,-78.952,-175.708,7.758,148.246
C06169=1228.020,395.975,-78.919,-175.709,7.756,148.245
C06170=1228.025,395.727,-78.885,-175.710,7.754,148.245
C06171=1228.029,395.480,-78.851,-175.711,7.751,148.244
C06172=1228.033,395.232,-78.816,-175.711,7.749,148.244
C06173=1228.037,394.984,-78.783,-175.712,7.746,148.244
C06174=1228.041,394.737,-78.749,-175.713,7.744,148.243
C06175=1228.045,394.489,-78.714,-175.714,7.741,148.243
C06176=1228.049,394.241,-78.681,-175.715,7.739,148.242
C06177=1228.053,393.994,-78.647,-175.716,7.736,148.242
C06178=1228.058,393.746,-78.613,-175.716,7.734,148.242
C06179=1228.062,393.465,-78.575,-175.717,7.731,148.241
C06180=1228.067,393.183,-78.535,-175.718,7.728,148.241
C06181=1228.072,392.902,-78.497,-175.719,7.725,148.240
C06182=1228.076,392.621,-78.459,-175.720,7.723,148.240
C06183=1228.080,392.373,-78.425,-175.721,7.720,148.239
C06184=1228.084,392.126,-78.391,-175.722,7.717,148.239
C06185=1228.088,391.877,-78.357,-175.722,7.715,148.238
C06186=1228.092,391.630,-78.324,-175.723,7.712,148.238
C06187=1228.097,391.382,-78.290,-175.724,7.710,148.238
C06188=1228.101,391.135,-78.256,-175.725,7.708,148.237
C06189=1228.104,390.887,-78.222,-175.726,7.706,148.237
C06190=1228.109,390.639,-78.188,-175.727,7.703,148.237
C06191=1228.112,390.392,-78.154,-175.727,7.701,148.236
C06192=1228.117,390.144,-78.121,-175.728,7.698,148.236
C06193=1228.121,389.896,-78.086,-175.729,7.695,148.235
C06194=1228.125,389.648,-78.053,-175.730,7.693,148.235
C06195=1228.129,389.401,-78.019,-175.731,7.690,148.234
C06196=1228.133,389.153,-77.985,-175.732,7.688,148.234
C06197=1228.137,388.906,-77.951,-175.733,7.685,148.234
C06198=1228.141,388.658,-77.918,-175.734,7.682,148.233
C06199=1228.146,388.410,-77.884,-175.735,7.680,148.233
C06200=1228.149,388.163,-77.850,-175.735,7.677,148.232
C06201=1228.154,387.915,-77.817,-175.737,7.674,148.232
C06202=1228.158,387.667,-77.783,-175.737,7.672,148.232
C06203=1228.162,387.419,-77.749,-175.738,7.670,148.231
C06204=1228.166,387.172,-77.715,-175.739,7.668,148.231
C06205=1228.170,386.924,-77.682,-175.740,7.665,148.230
C06206=1228.174,386.677,-77.648,-175.741,7.662,148.230
C06207=1228.178,386.429,-77.614,-175.742,7.660,148.230
C06208=1228.182,386.181,-77.581,-175.743,7.657,148.229
C06209=1228.186,385.933,-77.547,-175.744,7.654,148.229
C06210=1228.191,385.685,-77.513,-175.745,7.652,148.229
C06211=1228.195,385.438,-77.480,-175.746,7.650,148.228
C06212=1228.199,385.191,-77.446,-175.747,7.647,148.228
C06213=1228.203,384.943,-77.413,-175.748,7.645,148.227
C06214=1228.207,384.695,-77.378,-175.749,7.642,148.227
C06215=1228.211,384.447,-77.345,-175.750,7.639,148.227
C06216=1228.215,384.199,-77.312,-175.751,7.636,148.226
C06217=1228.219,383.952,-77.278,-175.752,7.634,148.226
C06218=1228.224,383.704,-77.244,-175.753,7.631,148.225
C06219=1228.228,383.456,-77.211,-175.754,7.628,148.225
C06220=1228.232,383.209,-77.178,-175.755,7.626,148.225
C06221=1228.235,382.961,-77.144,-175.756,7.624,148.224
C06222=1228.239,382.713,-77.111,-175.757,7.621,148.224
C06223=1228.244,382.465,-77.077,-175.758,7.618,148.223
C06224=1228.248,382.218,-77.043,-175.759,7.616,148.223
C06225=1228.252,381.970,-77.010,-175.760,7.613,148.223
C06226=1228.256,381.723,-76.977,-175.761,7.611,148.222
C06227=1228.260,381.475,-76.944,-175.763,7.608,148.222
C06228=1228.264,381.227,-76.909,-175.763,7.606,148.222
C06229=1228.269,380.979,-76.876,-175.764,7.603,148.221
C06230=1228.273,380.731,-76.842,-175.766,7.600,148.221
C06231=1228.277,380.483,-76.809,-175.767,7.597,148.220
C06232=1228.281,380.236,-76.776,-175.767,7.595,148.220
C06233=1228.285,379.989,-76.742,-175.769,7.593,148.220
C06234=1228.289,379.741,-76.709,-175.770,7.590,148.219
C06235=1228.293,379.493,-76.676,-175.771,7.587,148.219
C06236=1228.298,379.245,-76.642,-175.772,7.584,148.219
C06237=1228.302,378.997,-76.609,-175.773,7.582,148.218
C06238=1228.305,378.750,-76.575,-175.774,7.579,148.218
C06239=1228.309,378.502,-76.542,-175.776,7.577,148.218
C06240=1228.314,378.254,-76.508,-175.777,7.574,148.217
C06241=1228.318,378.006,-76.475,-175.778,7.571,148.217
C06242=1228.322,377.759,-76.442,-175.779,7.568,148.216
C06243=1228.326,377.511,-76.409,-175.780,7.566,148.216
C06244=1228.330,377.263,-76.376,-175.781,7.563,148.216
C06245=1228.334,377.016,-76.343,-175.782,7.561,148.215
C06246=1228.339,376.767,-76.309,-175.784,7.558,148.215
C06247=1228.343,376.520,-76.275,-175.785,7.555,148.215
C06248=1228.347,376.273,-76.242,-175.786,7.552,148.214
C06249=1228.351,376.025,-76.209,-175.787,7.550,148.214
C06250=1228.355,375.777,-76.176,-175.788,7.548,148.214
C06251=1228.360,375.529,-76.142,-175.789,7.545,148.213
C06252=1228.363,375.281,-76.109,-175.791,7.542,148.213
C06253=1228.367,375.033,-76.076,-175.792,7.539,148.213
C06254=1228.371,374.786,-76.043,-175.793,7.537,148.212
C06255=1228.376,374.538,-76.009,-175.794,7.534,148.212
C06256=1228.380,374.290,-75.976,-175.796,7.531,148.212
C06257=1228.384,374.042,-75.943,-175.797,7.528,148.211
C06258=1228.388,373.795,-75.910,-175.798,7.526,148.211
C06259=1228.392,373.547,-75.877,-175.799,7.523,148.210
C06260=1228.396,373.299,-75.844,-175.800,7.521,148.210
C06261=1228.400,373.051,-75.811,-175.801,7.518,148.210
C06262=1228.404,372.804,-75.777,-175.803,7.515,148.209
C06263=1228.409,372.556,-75.744,-175.804,7.513,148.209
C06264=1228.413,372.308,-75.711,-175.805,7.510,148.209
C06265=1228.417,372.061,-75.678,-175.807,7.507,148.208
C06266=1228.421,371.812,-75.645,-175.808,7.504,148.208
C06267=1228.425,371.564,-75.612,-175.809,7.502,148.208
C06268=1228.430,371.317,-75.579,-175.810,7.499,148.207
C06269=1228.434,371.069,-75.546,-175.812,7.496,148.207
C06270=1228.438,370.821,-75.513,-175.813,7.494,148.207
C06271=1228.441,370.574,-75.480,-175.814,7.491,148.206
C06272=1228.445,370.326,-75.447,-175.816,7.488,148.206
C06273=1228.450,370.078,-75.414,-175.817,7.486,148.206
C06274=1228.454,369.830,-75.382,-175.818,7.483,148.206
C06275=1228.458,369.582,-75.348,-175.820,7.480,148.205
C06276=1228.462,369.335,-75.315,-175.821,7.477,148.205
C06277=1228.466,369.087,-75.282,-175.822,7.475,148.205
C06278=1228.471,368.839,-75.249,-175.824,7.472,148.204
C06279=1228.475,368.591,-75.216,-175.825,7.469,148.204
C06280=1228.479,368.343,-75.183,-175.827,7.467,148.204
C06281=1228.483,368.096,-75.151,-175.828,7.464,148.203
C06282=1228.487,367.849,-75.118,-175.829,7.461,148.203
C06283=1228.492,367.569,-75.080,-175.831,7.459,148.203
C06284=1228.497,367.289,-75.044,-175.832,7.455,148.202
C06285=1228.501,367.009,-75.006,-175.834,7.452,148.202
C06286=1228.505,366.730,-74.969,-175.836,7.449,148.202
C06287=1228.510,366.482,-74.937,-175.837,7.446,148.201
C06288=1228.514,366.235,-74.904,-175.839,7.443,148.201
C06289=1228.519,365.987,-74.871,-175.840,7.440,148.201
C06290=1228.523,365.739,-74.838,-175.841,7.438,148.200
C06291=1228.526,365.491,-74.806,-175.843,7.435,148.200
C06292=1228.531,365.243,-74.773,-175.844,7.433,148.200
C06293=1228.535,364.995,-74.740,-175.846,7.430,148.200
C06294=1228.539,364.747,-74.707,-175.847,7.427,148.199
C06295=1228.543,364.500,-74.674,-175.849,7.425,148.199
C06296=1228.547,364.252,-74.642,-175.850,7.422,148.199
C06297=1228.551,364.004,-74.609,-175.851,7.419,148.199
C06298=1228.555,363.756,-74.576,-175.853,7.417,148.198
C06299=1228.560,363.508,-74.544,-175.854,7.414,148.198
C06300=1228.564,363.261,-74.511,-175.856,7.410,148.198
C06301=1228.568,363.013,-74.479,-175.857,7.408,148.197
C06302=1228.572,362.765,-74.445,-175.859,7.405,148.197
C06303=1228.576,362.517,-74.412,-175.860,7.402,148.197
C06304=1228.580,362.269,-74.380,-175.862,7.400,148.197
C06305=1228.584,362.021,-74.347,-175.864,7.397,148.196
C06306=1228.589,361.773,-74.315,-175.865,7.395,148.196
C06307=1228.592,361.526,-74.282,-175.866,7.392,148.196
C06308=1228.597,361.278,-74.250,-175.867,7.389,148.195
C06309=1228.601,361.030,-74.217,-175.870,7.386,148.195
C06310=1228.606,360.782,-74.185,-175.871,7.383,148.195
C06311=1228.609,360.535,-74.152,-175.872,7.380,148.195
C06312=1228.614,360.286,-74.120,-175.874,7.378,148.194
C06313=1228.618,360.038,-74.086,-175.876,7.375,148.194
C06314=1228.622,359.791,-74.055,-175.877,7.373,148.194
C06315=1228.626,359.543,-74.022,-175.878,7.370,148.194
C06316=1228.631,359.295,-73.989,-175.880,7.368,148.193
C06317=1228.634,359.048,-73.957,-175.882,7.364,148.193
C06318=1228.638,358.799,-73.924,-175.883,7.361,148.193
C06319=1228.643,358.551,-73.892,-175.885,7.359,148.193
C06320=1228.647,358.304,-73.860,-175.887,7.356,148.192
C06321=1228.651,358.056,-73.827,-175.888,7.354,148.192
C06322=1228.655,357.808,-73.795,-175.889,7.351,148.192
C06323=1228.659,357.560,-73.762,-175.892,7.348,148.192
C06324=1228.664,357.312,-73.730,-175.893,7.345,148.191
C06325=1228.668,357.065,-73.698,-175.895,7.343,148.191
C06326=1228.672,356.817,-73.665,-175.897,7.340,148.191
C06327=1228.676,356.569,-73.633,-175.898,7.337,148.191
C06328=1228.680,356.321,-73.600,-175.899,7.335,148.190
C06329=1228.684,356.073,-73.568,-175.901,7.331,148.190
C06330=1228.689,355.825,-73.536,-175.903,7.329,148.190
C06331=1228.693,355.577,-73.503,-175.905,7.326,148.190
C06332=1228.697,355.329,-73.471,-175.906,7.324,148.190
C06333=1228.701,355.081,-73.439,-175.908,7.321,148.189
C06334=1228.705,354.834,-73.407,-175.909,7.318,148.189
C06335=1228.709,354.586,-73.374,-175.911,7.315,148.189
C06336=1228.713,354.338,-73.342,-175.913,7.312,148.189
C06337=1228.718,354.090,-73.310,-175.915,7.310,148.188
C06338=1228.722,353.842,-73.278,-175.916,7.307,148.188
C06339=1228.726,353.595,-73.245,-175.918,7.305,148.188
C06340=1228.730,353.347,-73.213,-175.920,7.301,148.188
C06341=1228.734,353.098,-73.181,-175.922,7.299,148.188
C06342=1228.738,352.851,-73.150,-175.923,7.296,148.187
C06343=1228.743,352.602,-73.117,-175.924,7.294,148.187
C06344=1228.747,352.354,-73.085,-175.926,7.291,148.187
C06345=1228.751,352.107,-73.052,-175.928,7.288,148.187
C06346=1228.755,351.859,-73.021,-175.930,7.285,148.187
C06347=1228.760,351.611,-72.988,-175.931,7.283,148.186
C06348=1228.763,351.363,-72.956,-175.933,7.280,148.186
C06349=1228.768,351.115,-72.924,-175.935,7.278,148.186
C06350=1228.772,350.867,-72.892,-175.937,7.274,148.186
C06351=1228.776,350.619,-72.860,-175.939,7.272,148.186
C06352=1228.781,350.372,-72.829,-175.940,7.269,148.185
C06353=1228.784,350.124,-72.796,-175.942,7.267,148.185
C06354=1228.789,349.876,-72.764,-175.943,7.264,148.185
C06355=1228.793,349.629,-72.732,-175.946,7.261,148.185
C06356=1228.797,349.380,-72.700,-175.947,7.258,148.185
C06357=1228.801,349.132,-72.668,-175.949,7.256,148.184
C06358=1228.805,348.885,-72.636,-175.950,7.253,148.184
C06359=1228.810,348.636,-72.604,-175.953,7.250,148.184
C06360=1228.813,348.388,-72.572,-175.954,7.247,148.184
C06361=1228.819,348.141,-72.540,-175.956,7.245,148.184
C06362=1228.822,347.893,-72.508,-175.958,7.242,148.183
C06363=1228.826,347.645,-72.476,-175.959,7.240,148.183
C06364=1228.831,347.397,-72.444,-175.961,7.236,148.183
C06365=1228.835,347.149,-72.412,-175.963,7.234,148.183
C06366=1228.839,346.900,-72.381,-175.965,7.232,148.183
C06367=1228.844,346.653,-72.349,-175.967,7.229,148.183
C06368=1228.847,346.405,-72.317,-175.969,7.226,148.182
C06369=1228.852,346.157,-72.286,-175.970,7.223,148.182
C06370=1228.856,345.909,-72.253,-175.972,7.221,148.182
C06371=1228.860,345.661,-72.221,-175.974,7.218,148.182
C06372=1228.864,345.414,-72.190,-175.976,7.215,148.182
C06373=1228.869,345.165,-72.158,-175.978,7.212,148.182
C06374=1228.872,344.917,-72.126,-175.980,7.210,148.182
C06375=1228.877,344.669,-72.095,-175.981,7.207,148.181
C06376=1228.881,344.421,-72.063,-175.983,7.204,148.181
C06377=1228.886,344.174,-72.031,-175.985,7.201,148.181
C06378=1228.889,343.925,-71.999,-175.987,7.199,148.181
C06379=1228.894,343.678,-71.968,-175.989,7.197,148.181
C06380=1228.898,343.429,-71.937,-175.991,7.193,148.181
C06381=1228.902,343.181,-71.904,-175.993,7.191,148.180
C06382=1228.907,342.934,-71.873,-175.994,7.188,148.180
C06383=1228.910,342.686,-71.841,-175.996,7.186,148.180
C06384=1228.915,342.438,-71.809,-175.998,7.183,148.180
C06385=1228.919,342.189,-71.778,-176.000,7.180,148.180
C06386=1228.924,341.942,-71.746,-176.002,7.178,148.180
C06387=1228.928,341.665,-71.711,-176.004,7.174,148.179
C06388=1228.933,341.386,-71.676,-176.007,7.171,148.179
C06389=1228.937,341.109,-71.640,-176.008,7.169,148.179
C06390=1228.942,340.832,-71.605,-176.010,7.165,148.179
C06391=1228.947,340.583,-71.573,-176.012,7.163,148.179
C06392=1228.951,340.336,-71.542,-176.014,7.161,148.179
C06393=1228.955,340.088,-71.510,-176.016,7.157,148.179
C06394=1228.959,339.840,-71.479,-176.018,7.155,148.178
C06395=1228.963,339.592,-71.447,-176.020,7.152,148.178
C06396=1228.967,339.344,-71.416,-176.022,7.150,148.178
C06397=1228.971,339.096,-71.385,-176.024,7.146,148.178
C06398=1228.976,338.848,-71.352,-176.025,7.144,148.178
C06399=1228.980,338.599,-71.321,-176.027,7.142,148.178
C06400=1228.985,338.352,-71.290,-176.030,7.138,148.178
C06401=1228.989,338.103,-71.259,-176.031,7.136,148.178
C06402=1228.993,337.856,-71.227,-176.033,7.134,148.178
C06403=1228.997,337.607,-71.196,-176.035,7.131,148.177
C06404=1229.001,337.360,-71.165,-176.038,7.128,148.177
C06405=1229.005,337.111,-71.133,-176.039,7.125,148.177
C06406=1229.009,336.864,-71.102,-176.041,7.123,148.177
C06407=1229.014,336.615,-71.071,-176.044,7.120,148.177
C06408=1229.018,336.368,-71.039,-176.045,7.117,148.177
C06409=1229.022,336.119,-71.008,-176.047,7.115,148.177
C06410=1229.026,335.872,-70.977,-176.049,7.113,148.177
C06411=1229.030,335.623,-70.946,-176.051,7.109,148.176
C06412=1229.034,335.376,-70.914,-176.053,7.107,148.176
C06413=1229.038,335.127,-70.883,-176.055,7.104,148.176
C06414=1229.043,334.880,-70.852,-176.057,7.101,148.176
C06415=1229.047,334.632,-70.821,-176.059,7.099,148.176
C06416=1229.051,334.384,-70.790,-176.061,7.096,148.176
C06417=1229.056,334.136,-70.758,-176.063,7.094,148.176
C06418=1229.060,333.888,-70.727,-176.065,7.091,148.176
C06419=1229.064,333.640,-70.696,-176.067,7.089,148.176
C06420=1229.068,333.392,-70.664,-176.069,7.086,148.176
C06421=1229.073,333.144,-70.634,-176.071,7.083,148.176
C06422=1229.077,332.896,-70.602,-176.073,7.080,148.175
C06423=1229.081,332.648,-70.571,-176.075,7.078,148.175
C06424=1229.086,332.400,-70.540,-176.077,7.076,148.175
C06425=1229.089,332.152,-70.508,-176.079,7.072,148.175
C06426=1229.094,331.904,-70.478,-176.081,7.070,148.175
C06427=1229.099,331.656,-70.447,-176.083,7.068,148.175
C06428=1229.103,331.407,-70.416,-176.085,7.064,148.175
C06429=1229.107,331.160,-70.384,-176.087,7.062,148.175
C06430=1229.111,330.911,-70.353,-176.089,7.060,148.175
C06431=1229.115,330.663,-70.323,-176.091,7.057,148.175
C06432=1229.119,330.415,-70.292,-176.093,7.054,148.175
C06433=1229.123,330.167,-70.260,-176.095,7.052,148.175
C06434=1229.128,329.919,-70.230,-176.097,7.049,148.174
C06435=1229.132,329.671,-70.199,-176.100,7.046,148.174
C06436=1229.136,329.423,-70.168,-176.101,7.044,148.174
C06437=1229.141,329.175,-70.137,-176.103,7.042,148.174
C06438=1229.145,328.927,-70.107,-176.105,7.038,148.174
C06439=1229.148,328.679,-70.075,-176.108,7.036,148.174
C06440=1229.153,328.431,-70.044,-176.110,7.034,148.174
C06441=1229.158,328.183,-70.013,-176.111,7.031,148.174
C06442=1229.162,327.935,-69.982,-176.114,7.028,148.174
C06443=1229.166,327.687,-69.952,-176.116,7.026,148.174
C06444=1229.170,327.439,-69.921,-176.118,7.023,148.174
C06445=1229.174,327.190,-69.890,-176.120,7.020,148.174
C06446=1229.179,326.942,-69.860,-176.122,7.018,148.174
C06447=1229.183,326.694,-69.829,-176.124,7.016,148.174
C06448=1229.187,326.446,-69.798,-176.126,7.012,148.173
C06449=1229.191,326.199,-69.767,-176.128,7.010,148.174
C06450=1229.196,325.951,-69.736,-176.130,7.008,148.174
C06451=1229.200,325.703,-69.705,-176.132,7.005,148.173
C06452=1229.204,325.454,-69.675,-176.135,7.002,148.173
C06453=1229.208,325.206,-69.644,-176.137,7.000,148.173
C06454=1229.213,324.959,-69.613,-176.138,6.997,148.173
C06455=1229.216,324.710,-69.583,-176.141,6.994,148.173
C06456=1229.221,324.462,-69.553,-176.143,6.992,148.173
C06457=1229.226,324.214,-69.522,-176.145,6.990,148.173
C06458=1229.230,323.966,-69.491,-176.147,6.986,148.173
C06459=1229.233,323.717,-69.460,-176.149,6.984,148.173
C06460=1229.238,323.469,-69.430,-176.151,6.982,148.173
C06461=1229.243,323.221,-69.399,-176.153,6.980,148.173
C06462=1229.247,322.974,-69.369,-176.156,6.976,148.173
C06463=1229.251,322.725,-69.338,-176.158,6.974,148.173
C06464=1229.255,322.477,-69.307,-176.160,6.972,148.173
C06465=1229.259,322.229,-69.277,-176.162,6.969,148.173
C06466=1229.264,321.982,-69.246,-176.164,6.966,148.173
C06467=1229.267,321.733,-69.216,-176.166,6.964,148.173
C06468=1229.272,321.485,-69.185,-176.169,6.961,148.173
C06469=1229.276,321.237,-69.155,-176.171,6.959,148.173
C06470=1229.280,320.989,-69.124,-176.173,6.956,148.173
C06471=1229.285,320.741,-69.094,-176.175,6.953,148.173
C06472=1229.289,320.492,-69.064,-176.177,6.951,148.173
C06473=1229.293,320.244,-69.033,-176.179,6.949,148.173
C06474=1229.298,319.996,-69.002,-176.181,6.946,148.173
C06475=1229.302,319.749,-68.972,-176.184,6.943,148.173
C06476=1229.307,319.500,-68.942,-176.186,6.941,148.173
C06477=1229.310,319.252,-68.912,-176.188,6.938,148.173
C06478=1229.314,319.004,-68.881,-176.190,6.935,148.173
C06479=1229.318,318.756,-68.851,-176.192,6.933,148.173
C06480=1229.323,318.507,-68.821,-176.194,6.931,148.172
C06481=1229.327,318.260,-68.790,-176.197,6.928,148.172
C06482=1229.332,318.012,-68.760,-176.199,6.925,148.173
C06483=1229.335,317.763,-68.730,-176.201,6.923,148.173
C06484=1229.340,317.515,-68.699,-176.203,6.921,148.173
C06485=1229.344,317.267,-68.669,-176.206,6.918,148.173
C06486=1229.349,317.019,-68.639,-176.207,6.915,148.172
C06487=1229.353,316.771,-68.609,-176.209,6.913,148.172
C06488=1229.358,316.522,-68.579,-176.212,6.910,148.172
C06489=1229.361,316.275,-68.548,-176.214,6.908,148.173
C06490=1229.365,316.026,-68.517,-176.216,6.906,148.173
C06491=1229.370,315.751,-68.485,-176.219,6.903,148.173
C06492=1229.375,315.475,-68.450,-176.222,6.899,148.173
C06493=1229.379,315.199,-68.418,-176.224,6.897,148.173
C06494=1229.385,314.924,-68.384,-176.226,6.894,148.173
C06495=1229.389,314.675,-68.354,-176.228,6.892,148.173
C06496=1229.394,314.428,-68.323,-176.230,6.889,148.172
C06497=1229.397,314.179,-68.294,-176.233,6.886,148.172
C06498=1229.402,313.931,-68.263,-176.235,6.884,148.173
C06499=1229.406,313.682,-68.233,-176.237,6.882,148.173
C06500=1229.410,313.434,-68.204,-176.240,6.879,148.173
C06501=1229.415,313.186,-68.173,-176.242,6.877,148.173
C06502=1229.419,312.938,-68.144,-176.244,6.874,148.173
C06503=1229.423,312.690,-68.114,-176.246,6.871,148.173
C06504=1229.428,312.442,-68.083,-176.248,6.869,148.173
C06505=1229.432,312.194,-68.053,-176.251,6.867,148.173
C06506=1229.436,311.946,-68.024,-176.253,6.865,148.173
C06507=1229.441,311.697,-67.994,-176.255,6.862,148.173
C06508=1229.445,311.449,-67.964,-176.257,6.859,148.173
C06509=1229.449,311.201,-67.934,-176.260,6.857,148.173
C06510=1229.453,310.953,-67.903,-176.262,6.854,148.173
C06511=1229.458,310.705,-67.874,-176.264,6.852,148.173
C06512=1229.462,310.457,-67.844,-176.266,6.849,148.173
C06513=1229.467,310.208,-67.814,-176.268,6.847,148.173
C06514=1229.471,309.960,-67.784,-176.271,6.844,148.173
C06515=1229.475,309.712,-67.755,-176.273,6.842,148.173
C06516=1229.480,309.464,-67.725,-176.275,6.840,148.173
C06517=1229.484,309.216,-67.695,-176.278,6.837,148.173
C06518=1229.488,308.968,-67.665,-176.280,6.834,148.173
C06519=1229.492,308.719,-67.636,-176.282,6.832,148.173
C06520=1229.497,308.471,-67.606,-176.284,6.830,148.173
C06521=1229.501,308.223,-67.575,-176.286,6.827,148.173
C06522=1229.505,307.975,-67.546,-176.289,6.825,148.173
C06523=1229.509,307.727,-67.517,-176.291,6.822,148.173
C06524=1229.513,307.478,-67.487,-176.293,6.819,148.173
C06525=1229.518,307.230,-67.457,-176.295,6.817,148.173
C06526=1229.522,306.982,-67.427,-176.298,6.815,148.173
C06527=1229.526,306.734,-67.397,-176.300,6.813,148.174
C06528=1229.530,306.486,-67.368,-176.303,6.810,148.174
C06529=1229.535,306.237,-67.339,-176.305,6.808,148.174
C06530=1229.540,305.989,-67.309,-176.307,6.805,148.174
C06531=1229.544,305.741,-67.279,-176.309,6.803,148.174
C06532=1229.548,305.492,-67.250,-176.312,6.800,148.174
C06533=1229.552,305.244,-67.220,-176.314,6.798,148.174
C06534=1229.556,304.996,-67.190,-176.316,6.796,148.174
C06535=1229.560,304.748,-67.161,-176.319,6.793,148.174
C06536=1229.565,304.500,-67.130,-176.321,6.790,148.174
C06537=1229.570,304.252,-67.101,-176.323,6.788,148.174
C06538=1229.574,304.004,-67.072,-176.325,6.786,148.174
C06539=1229.578,303.755,-67.042,-176.328,6.783,148.174
C06540=1229.582,303.507,-67.013,-176.330,6.781,148.174
C06541=1229.587,303.259,-66.984,-176.332,6.779,148.174
C06542=1229.591,303.011,-66.954,-176.334,6.777,148.174
C06543=1229.595,302.762,-66.925,-176.337,6.774,148.174
C06544=1229.599,302.514,-66.895,-176.339,6.771,148.175
C06545=1229.603,302.266,-66.866,-176.341,6.769,148.175
C06546=1229.608,302.018,-66.837,-176.344,6.766,148.175
C06547=1229.612,301.770,-66.807,-176.346,6.764,148.175
C06548=1229.617,301.521,-66.778,-176.348,6.762,148.175
C06549=1229.622,301.273,-66.748,-176.351,6.760,148.175
C06550=1229.626,301.024,-66.719,-176.353,6.757,148.175
C06551=1229.630,300.776,-66.690,-176.355,6.754,148.175
C06552=1229.634,300.528,-66.660,-176.358,6.752,148.175
C06553=1229.639,300.280,-66.631,-176.360,6.750,148.175
C06554=1229.643,300.032,-66.602,-176.362,6.747,148.175
C06555=1229.647,299.784,-66.572,-176.364,6.745,148.175
C06556=1229.652,299.535,-66.543,-176.367,6.743,148.175
C06557=1229.655,299.287,-66.514,-176.369,6.741,148.176
C06558=1229.659,299.039,-66.485,-176.372,6.738,148.176
C06559=1229.664,298.791,-66.456,-176.374,6.735,148.176
C06560=1229.668,298.543,-66.426,-176.376,6.733,148.176
C06561=1229.673,298.294,-66.398,-176.379,6.731,148.176
C06562=1229.677,298.046,-66.368,-176.381,6.728,148.176
C06563=1229.681,297.797,-66.339,-176.383,6.726,148.176
C06564=1229.686,297.550,-66.310,-176.385,6.724,148.176
C06565=1229.691,297.301,-66.281,-176.388,6.721,148.176
C06566=1229.695,297.053,-66.252,-176.391,6.719,148.176
C06567=1229.699,296.804,-66.222,-176.393,6.717,148.176
C06568=1229.703,296.556,-66.193,-176.395,6.714,148.176
C06569=1229.708,296.308,-66.164,-176.397,6.712,148.177
C06570=1229.712,296.060,-66.135,-176.400,6.709,148.177
C06571=1229.716,295.812,-66.106,-176.402,6.707,148.177
C06572=1229.720,295.563,-66.077,-176.404,6.705,148.177
C06573=1229.725,295.315,-66.048,-176.406,6.703,148.177
C06574=1229.730,295.066,-66.019,-176.409,6.700,148.177
C06575=1229.734,294.818,-65.990,-176.412,6.698,148.177
C06576=1229.737,294.570,-65.961,-176.414,6.695,148.177
C06577=1229.742,294.322,-65.933,-176.416,6.693,148.177
C06578=1229.746,294.074,-65.903,-176.418,6.691,148.177
C06579=1229.751,293.825,-65.875,-176.421,6.688,148.178
C06580=1229.755,293.576,-65.845,-176.423,6.686,148.178
C06581=1229.759,293.329,-65.817,-176.425,6.684,148.178
C06582=1229.764,293.080,-65.788,-176.427,6.682,148.178
C06583=1229.768,292.832,-65.758,-176.431,6.679,148.178
C06584=1229.773,292.584,-65.730,-176.433,6.677,148.178
C06585=1229.777,292.336,-65.701,-176.435,6.674,148.178
C06586=1229.781,292.087,-65.672,-176.437,6.673,148.178
C06587=1229.785,291.839,-65.643,-176.440,6.670,148.178
C06588=1229.790,291.591,-65.615,-176.442,6.667,148.179
C06589=1229.794,291.342,-65.585,-176.444,6.665,148.179
C06590=1229.798,291.094,-65.557,-176.447,6.663,148.179
C06591=1229.803,290.845,-65.529,-176.449,6.661,148.179
C06592=1229.807,290.597,-65.499,-176.452,6.658,148.179
C06593=1229.811,290.349,-65.471,-176.454,6.656,148.179
C06594=1229.816,290.101,-65.442,-176.456,6.654,148.179
C06595=1229.821,289.827,-65.410,-176.459,6.651,148.179
C06596=1229.825,289.552,-65.379,-176.462,6.649,148.180
C06597=1229.830,289.278,-65.347,-176.464,6.646,148.180
C06598=1229.835,289.004,-65.315,-176.467,6.644,148.180
C06599=1229.839,288.756,-65.287,-176.469,6.642,148.180
C06600=1229.844,288.508,-65.258,-176.472,6.639,148.180
C06601=1229.849,288.259,-65.230,-176.474,6.637,148.180
C06602=1229.852,288.011,-65.201,-176.476,6.634,148.180
C06603=1229.857,287.762,-65.172,-176.479,6.633,148.181
C06604=1229.862,287.514,-65.144,-176.481,6.630,148.181
C06605=1229.865,287.266,-65.115,-176.484,6.627,148.181
C06606=1229.870,287.018,-65.087,-176.486,6.625,148.181
C06607=1229.874,286.770,-65.058,-176.488,6.623,148.181
C06608=1229.878,286.521,-65.030,-176.490,6.621,148.181
C06609=1229.883,286.273,-65.001,-176.493,6.619,148.181
C06610=1229.887,286.025,-64.972,-176.496,6.616,148.181
C06611=1229.892,285.776,-64.944,-176.498,6.614,148.181
C06612=1229.896,285.528,-64.916,-176.500,6.612,148.182
C06613=1229.900,285.279,-64.887,-176.503,6.610,148.182
C06614=1229.904,285.032,-64.859,-176.505,6.608,148.182
C06615=1229.909,284.783,-64.830,-176.508,6.605,148.182
C06616=1229.914,284.535,-64.802,-176.510,6.602,148.182
C06617=1229.918,284.286,-64.773,-176.512,6.601,148.182
C06618=1229.923,284.038,-64.745,-176.515,6.598,148.183
C06619=1229.927,283.789,-64.717,-176.517,6.596,148.183
C06620=1229.931,283.540,-64.688,-176.520,6.593,148.183
C06621=1229.935,283.292,-64.660,-176.522,6.591,148.183
C06622=1229.940,283.044,-64.631,-176.525,6.589,148.183
C06623=1229.944,282.796,-64.603,-176.527,6.587,148.183
C06624=1229.948,282.547,-64.574,-176.529,6.585,148.184
C06625=1229.953,282.300,-64.547,-176.531,6.583,148.184
C06626=1229.957,282.051,-64.519,-176.535,6.580,148.184
C06627=1229.962,281.803,-64.490,-176.537,6.578,148.184
C06628=1229.965,281.554,-64.462,-176.539,6.576,148.184
C06629=1229.970,281.306,-64.434,-176.541,6.574,148.184
C06630=1229.974,281.057,-64.406,-176.543,6.572,148.184
C06631=1229.979,280.809,-64.377,-176.546,6.570,148.185
C06632=1229.983,280.561,-64.349,-176.549,6.567,148.185
C06633=1229.987,280.313,-64.321,-176.551,6.565,148.185
C06634=1229.992,280.064,-64.293,-176.553,6.563,148.185
C06635=1229.996,279.816,-64.265,-176.556,6.561,148.185
C06636=1230.001,279.567,-64.236,-176.558,6.558,148.185
C06637=1230.005,279.319,-64.209,-176.561,6.557,148.186
C06638=1230.009,279.070,-64.181,-176.563,6.554,148.186
C06639=1230.014,278.822,-64.152,-176.565,6.551,148.186
C06640=1230.018,278.573,-64.124,-176.568,6.549,148.186
C06641=1230.022,278.325,-64.096,-176.570,6.547,148.186
C06642=1230.027,278.077,-64.068,-176.573,6.545,148.186
C06643=1230.031,277.829,-64.040,-176.575,6.543,148.186
C06644=1230.036,277.580,-64.013,-176.578,6.540,148.187
C06645=1230.040,277.331,-63.984,-176.580,6.538,148.187
C06646=1230.045,277.083,-63.956,-176.583,6.536,148.187
C06647=1230.048,276.835,-63.928,-176.585,6.534,148.187
C06648=1230.053,276.587,-63.900,-176.587,6.532,148.187
C06649=1230.058,276.339,-63.872,-176.590,6.530,148.187
C06650=1230.062,276.090,-63.845,-176.592,6.528,148.188
C06651=1230.066,275.842,-63.817,-176.595,6.525,148.188
C06652=1230.071,275.593,-63.788,-176.597,6.523,148.188
C06653=1230.075,275.344,-63.761,-176.600,6.521,148.188
C06654=1230.080,275.096,-63.733,-176.602,6.519,148.188
C06655=1230.083,274.848,-63.705,-176.604,6.517,148.189
C06656=1230.089,274.600,-63.677,-176.607,6.515,148.189
C06657=1230.093,274.350,-63.649,-176.609,6.513,148.189
C06658=1230.097,274.103,-63.622,-176.612,6.511,148.189
C06659=1230.101,273.855,-63.594,-176.615,6.508,148.189
C06660=1230.106,273.605,-63.566,-176.617,6.506,148.189
C06661=1230.110,273.357,-63.538,-176.619,6.504,148.190
C06662=1230.115,273.110,-63.510,-176.622,6.502,148.190
C06663=1230.119,272.860,-63.483,-176.624,6.500,148.190
C06664=1230.123,272.612,-63.455,-176.626,6.498,148.190
C06665=1230.128,272.363,-63.427,-176.629,6.496,148.191
C06666=1230.132,272.115,-63.399,-176.631,6.493,148.191
C06667=1230.137,271.867,-63.371,-176.634,6.491,148.191
C06668=1230.141,271.618,-63.344,-176.636,6.488,148.191
C06669=1230.145,271.370,-63.316,-176.639,6.487,148.191
C06670=1230.150,271.122,-63.289,-176.641,6.485,148.191
C06671=1230.154,270.873,-63.261,-176.644,6.482,148.192
C06672=1230.159,270.624,-63.233,-176.646,6.481,148.192
C06673=1230.163,270.376,-63.206,-176.648,6.478,148.192
C06674=1230.168,270.128,-63.179,-176.651,6.476,148.192
C06675=1230.172,269.879,-63.150,-176.654,6.473,148.192
C06676=1230.176,269.631,-63.123,-176.656,6.472,148.193
C06677=1230.181,269.383,-63.096,-176.659,6.470,148.193
C06678=1230.185,269.134,-63.068,-176.661,6.467,148.193
C06679=1230.189,268.886,-63.040,-176.663,6.466,148.193
C06680=1230.194,268.637,-63.013,-176.666,6.463,148.193
C06681=1230.198,268.389,-62.986,-176.668,6.461,148.194
C06682=1230.202,268.140,-62.958,-176.671,6.460,148.194
C06683=1230.207,267.892,-62.931,-176.673,6.457,148.194
C06684=1230.211,267.644,-62.903,-176.675,6.455,148.194
C06685=1230.216,267.395,-62.876,-176.678,6.453,148.194
C06686=1230.221,267.146,-62.848,-176.681,6.450,148.195
C06687=1230.225,266.898,-62.820,-176.683,6.449,148.195
C06688=1230.230,266.650,-62.793,-176.685,6.446,148.195
C06689=1230.234,266.401,-62.766,-176.688,6.444,148.195
C06690=1230.238,266.152,-62.738,-176.690,6.442,148.195
C06691=1230.243,265.904,-62.711,-176.693,6.440,148.196
C06692=1230.247,265.656,-62.685,-176.695,6.438,148.196
C06693=1230.251,265.408,-62.657,-176.698,6.436,148.196
C06694=1230.255,265.159,-62.629,-176.700,6.434,148.196
C06695=1230.260,264.910,-62.602,-176.703,6.432,148.197
C06696=1230.264,264.662,-62.575,-176.705,6.430,148.197
C06697=1230.269,264.414,-62.548,-176.707,6.428,148.197
C06698=1230.273,264.165,-62.520,-176.710,6.425,148.197
C06699=1230.278,263.892,-62.490,-176.713,6.423,148.197
C06700=1230.283,263.620,-62.460,-176.715,6.422,148.198
C06701=1230.287,263.347,-62.431,-176.718,6.419,148.198
C06702=1230.293,263.074,-62.401,-176.721,6.417,148.198
C06703=1230.297,262.826,-62.374,-176.723,6.415,148.198
C06704=1230.302,262.577,-62.347,-176.726,6.413,148.199
C06705=1230.306,262.329,-62.319,-176.728,6.411,148.199
C06706=1230.310,262.081,-62.292,-176.730,6.409,148.199
C06707=1230.314,261.832,-62.265,-176.733,6.407,148.199
C06708=1230.319,261.583,-62.238,-176.736,6.405,148.200
C06709=1230.324,261.335,-62.211,-176.738,6.403,148.200
C06710=1230.328,261.086,-62.184,-176.741,6.400,148.200
C06711=1230.333,260.838,-62.157,-176.744,6.398,148.200
C06712=1230.337,260.590,-62.130,-176.746,6.396,148.200
C06713=1230.341,260.341,-62.103,-176.748,6.394,148.201
C06714=1230.346,260.092,-62.076,-176.751,6.392,148.201
C06715=1230.350,259.844,-62.049,-176.753,6.390,148.201
C06716=1230.355,259.595,-62.022,-176.756,6.388,148.201
C06717=1230.358,259.347,-61.994,-176.758,6.386,148.202
C06718=1230.363,259.099,-61.967,-176.760,6.384,148.202
C06719=1230.368,258.850,-61.940,-176.763,6.382,148.202
C06720=1230.373,258.601,-61.914,-176.766,6.380,148.202
C06721=1230.377,258.353,-61.887,-176.768,6.378,148.202
C06722=1230.381,258.105,-61.860,-176.770,6.376,148.203
C06723=1230.385,257.855,-61.833,-176.773,6.374,148.203
C06724=1230.390,257.607,-61.806,-176.776,6.372,148.203
C06725=1230.395,257.358,-61.779,-176.778,6.370,148.203
C06726=1230.399,257.110,-61.752,-176.780,6.368,148.204
C06727=1230.403,256.862,-61.725,-176.783,6.366,148.204
C06728=1230.408,256.613,-61.698,-176.785,6.364,148.204
C06729=1230.412,256.365,-61.672,-176.788,6.362,148.204
C06730=1230.416,256.117,-61.645,-176.790,6.360,148.205
C06731=1230.421,255.868,-61.618,-176.793,6.358,148.205
C06732=1230.425,255.619,-61.592,-176.795,6.356,148.205
C06733=1230.430,255.371,-61.565,-176.798,6.354,148.205
C06734=1230.435,255.122,-61.538,-176.800,6.352,148.206
C06735=1230.439,254.874,-61.511,-176.803,6.351,148.206
C06736=1230.443,254.626,-61.484,-176.805,6.348,148.206
C06737=1230.448,254.377,-61.458,-176.807,6.346,148.206
C06738=1230.452,254.128,-61.432,-176.810,6.345,148.207
C06739=1230.457,253.880,-61.404,-176.813,6.343,148.207
C06740=1230.461,253.631,-61.377,-176.815,6.340,148.207
C06741=1230.465,253.383,-61.351,-176.818,6.338,148.207
C06742=1230.470,253.134,-61.325,-176.821,6.336,148.208
C06743=1230.474,252.886,-61.298,-176.823,6.334,148.208
C06744=1230.479,252.637,-61.271,-176.825,6.332,148.208
C06745=1230.484,252.388,-61.245,-176.828,6.330,148.208
C06746=1230.488,252.140,-61.218,-176.830,6.328,148.209
C06747=1230.492,251.892,-61.191,-176.833,6.326,148.209
C06748=1230.496,251.643,-61.165,-176.835,6.324,148.209
C06749=1230.501,251.394,-61.138,-176.838,6.322,148.209
C06750=1230.505,251.146,-61.112,-176.840,6.320,148.210
C06751=1230.510,250.897,-61.086,-176.843,6.318,148.210
C06752=1230.515,250.649,-61.058,-176.845,6.316,148.210
C06753=1230.519,250.400,-61.032,-176.848,6.314,148.210
C06754=1230.524,250.151,-61.006,-176.850,6.312,148.211
C06755=1230.528,249.903,-60.979,-176.853,6.310,148.211
C06756=1230.532,249.655,-60.952,-176.855,6.309,148.211
C06757=1230.537,249.406,-60.926,-176.857,6.307,148.211
C06758=1230.541,249.157,-60.899,-176.860,6.305,148.212
C06759=1230.545,248.908,-60.874,-176.862,6.303,148.212
C06760=1230.550,248.660,-60.847,-176.865,6.301,148.212
C06761=1230.554,248.411,-60.821,-176.867,6.299,148.212
C06762=1230.558,248.163,-60.794,-176.870,6.297,148.213
C06763=1230.564,247.915,-60.768,-176.872,6.295,148.213
C06764=1230.568,247.666,-60.742,-176.875,6.294,148.213
C06765=1230.573,247.417,-60.716,-176.878,6.292,148.214
C06766=1230.577,247.169,-60.689,-176.880,6.290,148.214
C06767=1230.582,246.920,-60.663,-176.882,6.288,148.214
C06768=1230.585,246.672,-60.636,-176.885,6.286,148.214
C06769=1230.590,246.423,-60.610,-176.888,6.284,148.215
C06770=1230.594,246.174,-60.583,-176.890,6.282,148.215
C06771=1230.599,245.926,-60.558,-176.892,6.280,148.215
C06772=1230.604,245.677,-60.532,-176.895,6.278,148.215
C06773=1230.608,245.429,-60.505,-176.898,6.276,148.216
C06774=1230.612,245.180,-60.479,-176.900,6.274,148.216
C06775=1230.617,244.932,-60.452,-176.903,6.272,148.216
C06776=1230.621,244.683,-60.427,-176.905,6.270,148.216
C06777=1230.626,244.434,-60.400,-176.907,6.268,148.217
C06778=1230.630,244.186,-60.374,-176.910,6.266,148.217
C06779=1230.635,243.938,-60.348,-176.913,6.264,148.217
C06780=1230.640,243.688,-60.322,-176.915,6.263,148.218
C06781=1230.644,243.440,-60.296,-176.918,6.261,148.218
C06782=1230.648,243.191,-60.270,-176.920,6.258,148.218
C06783=1230.653,242.942,-60.244,-176.923,6.257,148.218
C06784=1230.657,242.694,-60.217,-176.925,6.255,148.219
C06785=1230.662,242.446,-60.192,-176.928,6.253,148.219
C06786=1230.666,242.197,-60.166,-176.930,6.252,148.219
C06787=1230.671,241.948,-60.140,-176.933,6.250,148.220
C06788=1230.675,241.700,-60.113,-176.935,6.248,148.220
C06789=1230.679,241.451,-60.087,-176.937,6.246,148.220
C06790=1230.684,241.203,-60.062,-176.940,6.244,148.220
C06791=1230.689,240.954,-60.036,-176.943,6.242,148.221
C06792=1230.693,240.705,-60.010,-176.945,6.240,148.221
C06793=1230.697,240.457,-59.983,-176.948,6.238,148.221
C06794=1230.701,240.208,-59.958,-176.950,6.236,148.221
C06795=1230.707,239.960,-59.932,-176.952,6.234,148.222
C06796=1230.711,239.711,-59.906,-176.955,6.232,148.222
C06797=1230.715,239.462,-59.880,-176.958,6.230,148.222
C06798=1230.719,239.213,-59.854,-176.960,6.229,148.223
C06799=1230.725,238.965,-59.828,-176.963,6.227,148.223
C06800=1230.729,238.717,-59.802,-176.966,6.225,148.223
C06801=1230.733,238.468,-59.776,-176.968,6.223,148.223
C06802=1230.737,238.219,-59.751,-176.970,6.222,148.224
C06803=1230.743,237.948,-59.723,-176.973,6.219,148.224
C06804=1230.747,237.676,-59.695,-176.976,6.217,148.224
C06805=1230.752,237.405,-59.666,-176.979,6.215,148.225
C06806=1230.757,237.133,-59.638,-176.981,6.213,148.225
C06807=1230.761,236.885,-59.613,-176.984,6.212,148.225
C06808=1230.767,236.636,-59.587,-176.986,6.209,148.225
C06809=1230.771,236.387,-59.561,-176.989,6.208,148.226
C06810=1230.775,236.139,-59.535,-176.991,6.206,148.226
C06811=1230.780,235.891,-59.510,-176.994,6.204,148.226
C06812=1230.784,235.642,-59.484,-176.996,6.202,148.227
C06813=1230.789,235.393,-59.458,-176.999,6.200,148.227
C06814=1230.793,235.145,-59.433,-177.002,6.198,148.227
C06815=1230.798,234.896,-59.407,-177.004,6.197,148.228
C06816=1230.802,234.647,-59.381,-177.006,6.195,148.228
C06817=1230.807,234.399,-59.356,-177.009,6.193,148.228
C06818=1230.811,234.150,-59.330,-177.011,6.191,148.228
C06819=1230.816,233.901,-59.304,-177.014,6.189,148.229
C06820=1230.821,233.652,-59.279,-177.016,6.187,148.229
C06821=1230.825,233.404,-59.253,-177.019,6.186,148.229
C06822=1230.829,233.155,-59.228,-177.022,6.184,148.230
C06823=1230.834,232.907,-59.202,-177.024,6.182,148.230
C06824=1230.838,232.658,-59.177,-177.027,6.180,148.230
C06825=1230.843,232.409,-59.151,-177.029,6.179,148.231
C06826=1230.847,232.161,-59.125,-177.032,6.177,148.231
C06827=1230.852,231.912,-59.100,-177.034,6.175,148.231
C06828=1230.856,231.663,-59.075,-177.037,6.173,148.232
C06829=1230.861,231.415,-59.049,-177.039,6.171,148.232
C06830=1230.865,231.166,-59.024,-177.042,6.169,148.232
C06831=1230.870,230.918,-58.998,-177.044,6.167,148.232
C06832=1230.875,230.668,-58.973,-177.047,6.165,148.233
C06833=1230.878,230.420,-58.948,-177.049,6.164,148.233
C06834=1230.883,230.172,-58.923,-177.051,6.162,148.233
C06835=1230.887,229.922,-58.898,-177.054,6.161,148.234
C06836=1230.892,229.674,-58.872,-177.057,6.159,148.234
C06837=1230.897,229.425,-58.846,-177.059,6.157,148.234
C06838=1230.901,229.177,-58.821,-177.062,6.155,148.235
C06839=1230.906,228.928,-58.796,-177.065,6.153,148.235
C06840=1230.910,228.679,-58.770,-177.067,6.151,148.235
C06841=1230.915,228.431,-58.745,-177.070,6.149,148.236
C06842=1230.919,228.182,-58.720,-177.072,6.147,148.236
C06843=1230.924,227.934,-58.694,-177.074,6.146,148.236
C06844=1230.928,227.685,-58.669,-177.077,6.145,148.237
C06845=1230.932,227.436,-58.644,-177.080,6.143,148.237
C06846=1230.937,227.187,-58.619,-177.082,6.141,148.237
C06847=1230.942,226.938,-58.594,-177.085,6.139,148.238
C06848=1230.946,226.690,-58.568,-177.087,6.137,148.238
C06849=1230.951,226.441,-58.543,-177.090,6.135,148.238
C06850=1230.956,226.192,-58.518,-177.092,6.133,148.238
C06851=1230.959,225.944,-58.493,-177.094,6.132,148.239
C06852=1230.964,225.695,-58.468,-177.097,6.130,148.239
C06853=1230.969,225.446,-58.442,-177.100,6.128,148.239
C06854=1230.974,225.198,-58.418,-177.102,6.126,148.240
C06855=1230.978,224.949,-58.392,-177.105,6.124,148.240
C06856=1230.982,224.700,-58.368,-177.108,6.123,148.240
C06857=1230.987,224.452,-58.342,-177.110,6.121,148.241
C06858=1230.992,224.203,-58.318,-177.112,6.120,148.241
C06859=1230.996,223.954,-58.292,-177.115,6.118,148.241
C06860=1231.000,223.706,-58.268,-177.117,6.116,148.242
C06861=1231.005,223.457,-58.242,-177.120,6.114,148.242
C06862=1231.010,223.208,-58.217,-177.123,6.112,148.242
C06863=1231.014,222.959,-58.192,-177.125,6.110,148.243
C06864=1231.018,222.711,-58.167,-177.128,6.108,148.243
C06865=1231.023,222.462,-58.142,-177.130,6.107,148.243
C06866=1231.028,222.213,-58.117,-177.133,6.106,148.244
C06867=1231.032,221.964,-58.092,-177.135,6.104,148.244
C06868=1231.037,221.716,-58.068,-177.138,6.102,148.244
C06869=1231.042,221.468,-58.043,-177.141,6.100,148.245
C06870=1231.046,221.218,-58.017,-177.143,6.098,148.245
C06871=1231.050,220.970,-57.993,-177.145,6.097,148.245
C06872=1231.055,220.721,-57.968,-177.148,6.095,148.246
C06873=1231.060,220.472,-57.943,-177.150,6.093,148.246
C06874=1231.063,220.224,-57.918,-177.153,6.091,148.246
C06875=1231.068,219.975,-57.893,-177.156,6.090,148.247
C06876=1231.074,219.726,-57.869,-177.158,6.088,148.247
C06877=1231.077,219.477,-57.844,-177.161,6.086,148.247
C06878=1231.082,219.229,-57.819,-177.163,6.085,148.248
C06879=1231.087,218.980,-57.794,-177.166,6.083,148.248
C06880=1231.091,218.731,-57.770,-177.168,6.081,148.248
C06881=1231.096,218.482,-57.745,-177.171,6.079,148.249
C06882=1231.100,218.234,-57.720,-177.174,6.078,148.249
C06883=1231.105,217.985,-57.695,-177.177,6.076,148.250
C06884=1231.109,217.736,-57.670,-177.179,6.075,148.250
C06885=1231.114,217.487,-57.646,-177.181,6.073,148.250
C06886=1231.119,217.239,-57.621,-177.184,6.071,148.251
C06887=1231.122,216.990,-57.596,-177.187,6.069,148.251
C06888=1231.128,216.741,-57.571,-177.189,6.067,148.251
C06889=1231.132,216.493,-57.547,-177.192,6.065,148.252
C06890=1231.136,216.244,-57.522,-177.194,6.064,148.252
C06891=1231.141,215.995,-57.498,-177.197,6.063,148.252
C06892=1231.145,215.746,-57.473,-177.199,6.061,148.253
C06893=1231.150,215.497,-57.449,-177.202,6.059,148.253
C06894=1231.155,215.249,-57.424,-177.204,6.057,148.253
C06895=1231.159,215.000,-57.399,-177.207,6.055,148.254
C06896=1231.164,214.751,-57.375,-177.209,6.054,148.254
C06897=1231.169,214.503,-57.350,-177.212,6.052,148.254
C06898=1231.173,214.254,-57.326,-177.214,6.050,148.255
C06899=1231.177,214.005,-57.301,-177.217,6.048,148.255
C06900=1231.182,213.756,-57.277,-177.220,6.047,148.255
C06901=1231.186,213.508,-57.253,-177.222,6.046,148.256
C06902=1231.191,213.259,-57.228,-177.225,6.044,148.256
C06903=1231.195,213.010,-57.204,-177.227,6.042,148.257
C06904=1231.200,212.761,-57.179,-177.230,6.040,148.257
C06905=1231.204,212.512,-57.155,-177.233,6.038,148.257
C06906=1231.209,212.264,-57.130,-177.235,6.037,148.258
C06907=1231.214,211.994,-57.104,-177.238,6.035,148.258
C06908=1231.219,211.723,-57.078,-177.241,6.033,148.258
C06909=1231.224,211.452,-57.051,-177.244,6.031,148.259
C06910=1231.229,211.182,-57.024,-177.246,6.029,148.259
C06911=1231.233,210.934,-57.000,-177.248,6.028,148.259
C06912=1231.238,210.685,-56.975,-177.251,6.027,148.260
C06913=1231.242,210.436,-56.951,-177.254,6.025,148.260
C06914=1231.247,210.187,-56.927,-177.256,6.023,148.260
C06915=1231.252,209.938,-56.903,-177.259,6.021,148.261
C06916=1231.256,209.690,-56.879,-177.261,6.020,148.261
C06917=1231.261,209.440,-56.854,-177.264,6.018,148.262
C06918=1231.265,209.192,-56.830,-177.267,6.017,148.262
C06919=1231.270,208.943,-56.805,-177.269,6.015,148.262
C06920=1231.275,208.695,-56.781,-177.271,6.014,148.263
C06921=1231.280,208.445,-56.757,-177.274,6.012,148.263
C06922=1231.283,208.196,-56.733,-177.277,6.010,148.263
C06923=1231.289,207.948,-56.708,-177.279,6.008,148.264
C06924=1231.293,207.699,-56.684,-177.282,6.006,148.264
C06925=1231.298,207.450,-56.661,-177.284,6.005,148.264
C06926=1231.302,207.202,-56.637,-177.287,6.003,148.265
C06927=1231.307,206.952,-56.612,-177.290,6.002,148.265
C06928=1231.311,206.704,-56.588,-177.292,6.000,148.266
C06929=1231.316,206.455,-56.564,-177.295,5.999,148.266
C06930=1231.321,206.206,-56.540,-177.297,5.997,148.266
C06931=1231.325,205.958,-56.516,-177.300,5.995,148.267
C06932=1231.330,205.709,-56.492,-177.302,5.993,148.267
C06933=1231.334,205.460,-56.468,-177.305,5.992,148.267
C06934=1231.338,205.211,-56.444,-177.307,5.990,148.268
C06935=1231.343,204.963,-56.419,-177.310,5.989,148.268
C06936=1231.348,204.713,-56.396,-177.313,5.987,148.269
C06937=1231.352,204.465,-56.372,-177.315,5.986,148.269
C06938=1231.357,204.217,-56.348,-177.318,5.984,148.269
C06939=1231.362,203.967,-56.323,-177.320,5.982,148.270
C06940=1231.366,203.718,-56.299,-177.323,5.980,148.270
C06941=1231.371,203.469,-56.276,-177.325,5.979,148.270
C06942=1231.375,203.221,-56.252,-177.328,5.978,148.271
C06943=1231.379,202.972,-56.228,-177.330,5.976,148.271
C06944=1231.384,202.723,-56.204,-177.333,5.974,148.272
C06945=1231.389,202.475,-56.180,-177.335,5.973,148.272
C06946=1231.394,202.226,-56.156,-177.338,5.971,148.272
C06947=1231.398,201.976,-56.132,-177.341,5.969,148.273
C06948=1231.402,201.727,-56.108,-177.343,5.968,148.273
C06949=1231.407,201.479,-56.084,-177.345,5.967,148.273
C06950=1231.412,201.230,-56.061,-177.348,5.965,148.274
C06951=1231.416,200.982,-56.037,-177.351,5.963,148.274
C06952=1231.421,200.733,-56.014,-177.354,5.961,148.275
C06953=1231.426,200.484,-55.989,-177.356,5.960,148.275
C06954=1231.430,200.235,-55.966,-177.359,5.958,148.275
C06955=1231.435,199.986,-55.942,-177.361,5.957,148.276
C06956=1231.440,199.737,-55.918,-177.363,5.956,148.276
C06957=1231.444,199.489,-55.894,-177.366,5.954,148.276
C06958=1231.449,199.240,-55.871,-177.369,5.952,148.277
C06959=1231.453,198.991,-55.847,-177.372,5.950,148.277
C06960=1231.457,198.742,-55.823,-177.374,5.949,148.278
C06961=1231.462,198.493,-55.800,-177.376,5.947,148.278
C06962=1231.466,198.244,-55.775,-177.379,5.946,148.278
C06963=1231.471,197.995,-55.752,-177.381,5.945,148.279
C06964=1231.476,197.746,-55.729,-177.384,5.943,148.279
C06965=1231.480,197.498,-55.705,-177.387,5.941,148.280
C06966=1231.485,197.249,-55.681,-177.389,5.939,148.280
C06967=1231.489,197.000,-55.658,-177.392,5.938,148.280
C06968=1231.494,196.751,-55.634,-177.394,5.936,148.281
C06969=1231.498,196.502,-55.611,-177.397,5.935,148.281
C06970=1231.503,196.253,-55.587,-177.399,5.934,148.282
C06971=1231.508,196.005,-55.563,-177.402,5.932,148.282
C06972=1231.512,195.756,-55.540,-177.405,5.930,148.282
C06973=1231.517,195.507,-55.516,-177.407,5.929,148.283
C06974=1231.522,195.258,-55.493,-177.409,5.927,148.283
C06975=1231.526,195.009,-55.469,-177.412,5.925,148.283
C06976=1231.531,194.760,-55.446,-177.415,5.924,148.284
C06977=1231.535,194.511,-55.422,-177.417,5.923,148.284
C06978=1231.540,194.262,-55.399,-177.420,5.921,148.285
C06979=1231.545,194.013,-55.376,-177.423,5.919,148.285
C06980=1231.549,193.765,-55.351,-177.425,5.918,148.285
C06981=1231.554,193.516,-55.328,-177.428,5.917,148.286
C06982=1231.559,193.268,-55.306,-177.430,5.915,148.286
C06983=1231.563,193.019,-55.282,-177.432,5.914,148.287
C06984=1231.568,192.770,-55.259,-177.435,5.912,148.287
C06985=1231.572,192.521,-55.235,-177.438,5.910,148.287
C06986=1231.577,192.272,-55.212,-177.440,5.909,148.288
C06987=1231.582,192.023,-55.188,-177.443,5.908,148.288
C06988=1231.586,191.774,-55.165,-177.446,5.906,148.289
C06989=1231.591,191.525,-55.141,-177.448,5.905,148.289
C06990=1231.595,191.276,-55.119,-177.450,5.903,148.289
C06991=1231.600,191.027,-55.095,-177.453,5.901,148.290
C06992=1231.604,190.778,-55.072,-177.456,5.900,148.290
C06993=1231.609,190.529,-55.049,-177.458,5.898,148.291
C06994=1231.614,190.280,-55.025,-177.461,5.897,148.291
C06995=1231.619,190.032,-55.002,-177.463,5.896,148.291
C06996=1231.623,189.783,-54.980,-177.466,5.894,148.292
C06997=1231.628,189.534,-54.956,-177.469,5.892,148.292
C06998=1231.633,189.285,-54.933,-177.471,5.891,148.293
C06999=1231.637,189.036,-54.909,-177.473,5.889,148.293
C07000=1231.642,188.787,-54.886,-177.476,5.887,148.293
C07001=1231.646,188.538,-54.863,-177.479,5.887,148.294
C07002=1231.651,188.289,-54.840,-177.481,5.885,148.294
C07003=1231.655,188.040,-54.817,-177.483,5.884,148.295
C07004=1231.661,187.792,-54.794,-177.486,5.882,148.295
C07005=1231.665,187.543,-54.771,-177.489,5.881,148.296
C07006=1231.669,187.294,-54.747,-177.491,5.880,148.296
C07007=1231.674,187.045,-54.724,-177.494,5.878,148.296
C07008=1231.678,186.796,-54.701,-177.496,5.876,148.297
C07009=1231.683,186.547,-54.678,-177.499,5.875,148.297
C07010=1231.688,186.299,-54.655,-177.502,5.873,148.298
C07011=1231.693,186.029,-54.630,-177.504,5.871,148.298
C07012=1231.697,185.759,-54.605,-177.507,5.870,148.299
C07013=1231.703,185.489,-54.580,-177.510,5.869,148.299
C07014=1231.708,185.220,-54.555,-177.512,5.867,148.299
C07015=1231.712,184.971,-54.532,-177.515,5.866,148.300
C07016=1231.717,184.723,-54.509,-177.518,5.864,148.300
C07017=1231.722,184.474,-54.486,-177.520,5.863,148.301
C07018=1231.726,184.225,-54.463,-177.523,5.861,148.301
C07019=1231.731,183.975,-54.441,-177.525,5.860,148.302
C07020=1231.736,183.726,-54.417,-177.528,5.858,148.302
C07021=1231.740,183.478,-54.395,-177.531,5.856,148.302
C07022=1231.745,183.229,-54.371,-177.533,5.855,148.303
C07023=1231.749,182.980,-54.349,-177.536,5.854,148.303
C07024=1231.754,182.731,-54.326,-177.538,5.852,148.304
C07025=1231.759,182.482,-54.303,-177.541,5.851,148.304
C07026=1231.763,182.234,-54.280,-177.543,5.849,148.304
C07027=1231.768,181.984,-54.258,-177.546,5.849,148.305
C07028=1231.772,181.735,-54.235,-177.548,5.847,148.305
C07029=1231.777,181.486,-54.212,-177.551,5.845,148.306
C07030=1231.782,181.238,-54.190,-177.553,5.844,148.306
C07031=1231.786,180.989,-54.166,-177.556,5.842,148.307
C07032=1231.791,180.740,-54.143,-177.558,5.841,148.307
C07033=1231.796,180.491,-54.121,-177.561,5.839,148.307
C07034=1231.801,180.242,-54.098,-177.564,5.838,148.308
C07035=1231.804,179.993,-54.075,-177.566,5.837,148.308
C07036=1231.809,179.744,-54.053,-177.569,5.835,148.309
C07037=1231.814,179.496,-54.030,-177.571,5.834,148.309
C07038=1231.819,179.246,-54.007,-177.574,5.833,148.310
C07039=1231.823,178.997,-53.985,-177.576,5.832,148.310
C07040=1231.828,178.748,-53.962,-177.579,5.830,148.310
C07041=1231.833,178.499,-53.940,-177.581,5.828,148.311
C07042=1231.837,178.250,-53.916,-177.584,5.827,148.311
C07043=1231.842,178.001,-53.894,-177.587,5.825,148.312
C07044=1231.847,177.753,-53.871,-177.589,5.824,148.312
C07045=1231.851,177.504,-53.849,-177.592,5.823,148.313
C07046=1231.856,177.254,-53.826,-177.595,5.821,148.313
C07047=1231.860,177.006,-53.804,-177.597,5.820,148.313
C07048=1231.865,176.757,-53.781,-177.599,5.818,148.314
C07049=1231.869,176.508,-53.758,-177.602,5.817,148.314
C07050=1231.874,176.259,-53.737,-177.605,5.816,148.315
C07051=1231.879,176.010,-53.713,-177.607,5.815,148.315
C07052=1231.883,175.761,-53.691,-177.610,5.813,148.316
C07053=1231.889,175.512,-53.669,-177.612,5.811,148.316
C07054=1231.893,175.263,-53.646,-177.615,5.810,148.316
C07055=1231.898,175.014,-53.623,-177.617,5.808,148.317
C07056=1231.902,174.766,-53.601,-177.620,5.808,148.317
C07057=1231.907,174.516,-53.579,-177.622,5.806,148.318
C07058=1231.911,174.267,-53.556,-177.625,5.805,148.318
C07059=1231.916,174.019,-53.534,-177.628,5.803,148.319
C07060=1231.920,173.769,-53.512,-177.630,5.802,148.319
C07061=1231.926,173.521,-53.489,-177.632,5.801,148.320
C07062=1231.930,173.272,-53.467,-177.636,5.799,148.320
C07063=1231.934,173.022,-53.445,-177.638,5.798,148.320
C07064=1231.940,172.774,-53.422,-177.640,5.796,148.321
C07065=1231.944,172.525,-53.400,-177.643,5.796,148.321
C07066=1231.949,172.276,-53.378,-177.646,5.794,148.322
C07067=1231.953,172.027,-53.355,-177.648,5.793,148.322
C07068=1231.958,171.778,-53.333,-177.651,5.791,148.323
C07069=1231.963,171.529,-53.311,-177.653,5.790,148.323
C07070=1231.967,171.280,-53.288,-177.655,5.788,148.324
C07071=1231.972,171.031,-53.266,-177.658,5.787,148.324
C07072=1231.976,170.782,-53.244,-177.661,5.786,148.324
C07073=1231.982,170.533,-53.222,-177.663,5.785,148.325
C07074=1231.986,170.284,-53.199,-177.665,5.783,148.325
C07075=1231.990,170.035,-53.177,-177.669,5.781,148.326
C07076=1231.995,169.786,-53.155,-177.671,5.780,148.326
C07077=1232.000,169.537,-53.133,-177.673,5.779,148.327
C07078=1232.005,169.289,-53.110,-177.676,5.778,148.327
C07079=1232.009,169.039,-53.088,-177.679,5.776,148.328
C07080=1232.014,168.791,-53.066,-177.681,5.775,148.328
C07081=1232.019,168.541,-53.044,-177.684,5.774,148.329
C07082=1232.024,168.292,-53.022,-177.686,5.773,148.329
C07083=1232.028,168.044,-52.999,-177.689,5.771,148.329
C07084=1232.032,167.795,-52.978,-177.691,5.770,148.330
C07085=1232.037,167.546,-52.956,-177.694,5.768,148.330
C07086=1232.042,167.297,-52.933,-177.696,5.768,148.331
C07087=1232.047,167.047,-52.911,-177.699,5.766,148.331
C07088=1232.051,166.799,-52.890,-177.701,5.765,148.332
C07089=1232.056,166.549,-52.867,-177.704,5.763,148.332
C07090=1232.061,166.301,-52.846,-177.706,5.762,148.333
C07091=1232.066,166.051,-52.823,-177.709,5.760,148.333
C07092=1232.070,165.803,-52.801,-177.712,5.760,148.334
C07093=1232.074,165.554,-52.779,-177.714,5.758,148.334
C07094=1232.079,165.305,-52.757,-177.716,5.757,148.334
C07095=1232.084,165.056,-52.735,-177.720,5.755,148.335
C07096=1232.088,164.807,-52.713,-177.722,5.754,148.335
C07097=1232.093,164.558,-52.691,-177.724,5.753,148.336
C07098=1232.098,164.309,-52.670,-177.727,5.752,148.336
C07099=1232.103,164.059,-52.647,-177.730,5.750,148.337
C07100=1232.107,163.811,-52.625,-177.732,5.749,148.337
C07101=1232.112,163.561,-52.603,-177.735,5.748,148.338
C07102=1232.117,163.313,-52.582,-177.737,5.747,148.338
C07103=1232.121,163.063,-52.559,-177.740,5.745,148.339
C07104=1232.126,162.815,-52.538,-177.742,5.744,148.339
C07105=1232.131,162.566,-52.516,-177.745,5.742,148.339
C07106=1232.135,162.316,-52.495,-177.747,5.742,148.340
C07107=1232.140,162.068,-52.473,-177.750,5.740,148.340
C07108=1232.144,161.818,-52.451,-177.753,5.739,148.341
C07109=1232.149,161.570,-52.429,-177.755,5.737,148.341
C07110=1232.153,161.320,-52.407,-177.757,5.736,148.342
C07111=1232.158,161.072,-52.386,-177.760,5.735,148.342
C07112=1232.163,160.823,-52.364,-177.763,5.734,148.343
C07113=1232.167,160.574,-52.342,-177.765,5.732,148.343
C07114=1232.172,160.325,-52.320,-177.768,5.731,148.344
C07115=1232.178,160.056,-52.297,-177.770,5.729,148.344
C07116=1232.183,159.786,-52.274,-177.773,5.729,148.345
C07117=1232.188,159.518,-52.250,-177.776,5.727,148.345
C07118=1232.193,159.248,-52.226,-177.779,5.725,148.346
C07119=1232.198,158.999,-52.205,-177.781,5.725,148.346
C07120=1232.202,158.751,-52.183,-177.784,5.723,148.347
C07121=1232.207,158.501,-52.162,-177.786,5.722,148.347
C07122=1232.212,158.252,-52.140,-177.789,5.721,148.348
C07123=1232.217,158.003,-52.118,-177.791,5.719,148.348
C07124=1232.221,157.754,-52.096,-177.794,5.719,148.349
C07125=1232.226,157.505,-52.075,-177.797,5.717,148.349
C07126=1232.231,157.256,-52.054,-177.799,5.716,148.349
C07127=1232.235,157.007,-52.032,-177.802,5.714,148.350
C07128=1232.239,156.758,-52.010,-177.804,5.713,148.350
C07129=1232.245,156.509,-51.989,-177.807,5.712,148.351
C07130=1232.249,156.260,-51.967,-177.809,5.711,148.351
C07131=1232.254,156.011,-51.946,-177.812,5.709,148.352
C07132=1232.259,155.762,-51.925,-177.815,5.708,148.352
C07133=1232.263,155.513,-51.903,-177.817,5.707,148.353
C07134=1232.268,155.264,-51.881,-177.820,5.706,148.353
C07135=1232.273,155.015,-51.860,-177.822,5.705,148.354
C07136=1232.277,154.766,-51.839,-177.825,5.703,148.354
C07137=1232.282,154.517,-51.817,-177.827,5.702,148.355
C07138=1232.287,154.268,-51.796,-177.830,5.701,148.355
C07139=1232.291,154.018,-51.774,-177.832,5.700,148.356
C07140=1232.296,153.770,-51.752,-177.835,5.699,148.356
C07141=1232.301,153.520,-51.731,-177.838,5.698,148.357
C07142=1232.305,153.272,-51.710,-177.840,5.697,148.357
C07143=1232.310,153.022,-51.689,-177.842,5.695,148.357
C07144=1232.315,152.774,-51.667,-177.845,5.694,148.358
C07145=1232.320,152.524,-51.646,-177.848,5.692,148.358
C07146=1232.325,152.276,-51.624,-177.850,5.692,148.359
C07147=1232.329,152.026,-51.603,-177.852,5.691,148.359
C07148=1232.333,151.777,-51.582,-177.856,5.689,148.360
C07149=1232.338,151.529,-51.560,-177.858,5.688,148.360
C07150=1232.343,151.279,-51.539,-177.860,5.686,148.361
C07151=1232.348,151.030,-51.517,-177.863,5.686,148.361
C07152=1232.352,150.781,-51.497,-177.865,5.685,148.362
C07153=1232.357,150.532,-51.476,-177.868,5.683,148.362
C07154=1232.362,150.283,-51.454,-177.870,5.682,148.363
C07155=1232.367,150.033,-51.433,-177.873,5.681,148.363
C07156=1232.371,149.785,-51.412,-177.876,5.680,148.364
C07157=1232.376,149.536,-51.391,-177.879,5.678,148.364
C07158=1232.381,149.287,-51.369,-177.881,5.677,148.365
C07159=1232.386,149.037,-51.348,-177.883,5.676,148.365
C07160=1232.390,148.789,-51.327,-177.886,5.675,148.366
C07161=1232.395,148.540,-51.306,-177.888,5.674,148.366
C07162=1232.400,148.290,-51.285,-177.891,5.672,148.367
C07163=1232.404,148.042,-51.264,-177.893,5.671,148.367
C07164=1232.409,147.792,-51.243,-177.896,5.671,148.368
C07165=1232.414,147.543,-51.222,-177.899,5.669,148.368
C07166=1232.418,147.294,-51.200,-177.901,5.668,148.369
C07167=1232.423,147.045,-51.179,-177.903,5.667,148.369
C07168=1232.428,146.796,-51.159,-177.907,5.666,148.370
C07169=1232.433,146.548,-51.137,-177.909,5.665,148.370
C07170=1232.437,146.298,-51.116,-177.912,5.663,148.371
C07171=1232.442,146.048,-51.095,-177.914,5.662,148.371
C07172=1232.446,145.800,-51.074,-177.916,5.661,148.372
C07173=1232.452,145.551,-51.053,-177.919,5.660,148.372
C07174=1232.456,145.302,-51.033,-177.921,5.659,148.373
C07175=1232.461,145.053,-51.011,-177.924,5.657,148.373
C07176=1232.465,144.803,-50.990,-177.927,5.656,148.374
C07177=1232.470,144.554,-50.969,-177.929,5.656,148.374
C07178=1232.475,144.305,-50.948,-177.932,5.654,148.375
C07179=1232.479,144.057,-50.927,-177.934,5.653,148.375
C07180=1232.484,143.807,-50.906,-177.936,5.652,148.376
C07181=1232.489,143.558,-50.886,-177.940,5.651,148.376
C07182=1232.494,143.309,-50.865,-177.942,5.650,148.377
C07183=1232.499,143.060,-50.844,-177.945,5.648,148.377
C07184=1232.503,142.811,-50.823,-177.947,5.647,148.378
C07185=1232.508,142.562,-50.802,-177.950,5.646,148.378
C07186=1232.512,142.313,-50.781,-177.952,5.645,148.379
C07187=1232.517,142.063,-50.760,-177.955,5.644,148.379
C07188=1232.522,141.814,-50.740,-177.957,5.643,148.380
C07189=1232.527,141.565,-50.719,-177.960,5.642,148.380
C07190=1232.532,141.316,-50.699,-177.962,5.641,148.381
C07191=1232.536,141.068,-50.677,-177.965,5.640,148.381
C07192=1232.541,140.819,-50.656,-177.968,5.638,148.382
C07193=1232.546,140.569,-50.636,-177.970,5.637,148.382
C07194=1232.550,140.320,-50.615,-177.972,5.636,148.383
C07195=1232.556,140.071,-50.594,-177.975,5.635,148.383
C07196=1232.559,139.822,-50.573,-177.977,5.634,148.384
C07197=1232.565,139.572,-50.552,-177.980,5.633,148.384
C07198=1232.569,139.323,-50.532,-177.983,5.631,148.385
C07199=1232.574,139.074,-50.511,-177.985,5.631,148.385
C07200=1232.579,138.825,-50.491,-177.988,5.629,148.386
C07201=1232.583,138.576,-50.470,-177.991,5.628,148.386
C07202=1232.588,138.327,-50.449,-177.993,5.627,148.387
C07203=1232.593,138.078,-50.429,-177.996,5.626,148.387
C07204=1232.598,137.829,-50.408,-177.998,5.625,148.388
C07205=1232.602,137.580,-50.388,-178.001,5.624,148.388
C07206=1232.608,137.330,-50.367,-178.003,5.622,148.389
C07207=1232.612,137.082,-50.346,-178.006,5.622,148.389
C07208=1232.616,136.833,-50.326,-178.008,5.621,148.390
C07209=1232.622,136.583,-50.305,-178.011,5.619,148.391
C07210=1232.626,136.334,-50.285,-178.013,5.618,148.391
C07211=1232.630,136.085,-50.264,-178.016,5.618,148.392
C07212=1232.636,135.836,-50.243,-178.018,5.617,148.392
C07213=1232.640,135.587,-50.223,-178.021,5.615,148.393
C07214=1232.645,135.338,-50.202,-178.024,5.615,148.393
C07215=1232.650,135.089,-50.182,-178.026,5.614,148.394
C07216=1232.654,134.839,-50.162,-178.029,5.612,148.394
C07217=1232.660,134.590,-50.141,-178.031,5.611,148.395
C07218=1232.664,134.341,-50.121,-178.034,5.611,148.395
C07219=1232.669,134.073,-50.098,-178.036,5.609,148.396
C07220=1232.674,133.804,-50.077,-178.039,5.608,148.396
C07221=1232.679,133.535,-50.054,-178.042,5.607,148.397
C07222=1232.685,133.266,-50.033,-178.045,5.606,148.397
C07223=1232.689,133.017,-50.012,-178.047,5.604,148.398
C07224=1232.694,132.768,-49.992,-178.050,5.603,148.399
C07225=1232.699,132.519,-49.971,-178.052,5.603,148.399
C07226=1232.703,132.270,-49.951,-178.055,5.601,148.400
C07227=1232.708,132.021,-49.931,-178.057,5.600,148.400
C07228=1232.714,131.772,-49.910,-178.060,5.599,148.401
C07229=1232.718,131.523,-49.890,-178.062,5.598,148.401
C07230=1232.723,131.274,-49.870,-178.065,5.597,148.402
C07231=1232.727,131.025,-49.850,-178.068,5.596,148.402
C07232=1232.732,130.775,-49.829,-178.070,5.595,148.403
C07233=1232.737,130.526,-49.809,-178.073,5.594,148.403
C07234=1232.741,130.277,-49.788,-178.075,5.593,148.404
C07235=1232.746,130.028,-49.769,-178.078,5.592,148.404
C07236=1232.751,129.779,-49.748,-178.081,5.590,148.405
C07237=1232.756,129.530,-49.727,-178.083,5.590,148.405
C07238=1232.760,129.280,-49.708,-178.085,5.589,148.406
C07239=1232.765,129.032,-49.688,-178.088,5.588,148.406
C07240=1232.770,128.783,-49.667,-178.091,5.587,148.407
C07241=1232.775,128.533,-49.648,-178.093,5.586,148.407
C07242=1232.780,128.284,-49.627,-178.096,5.585,148.408
C07243=1232.784,128.035,-49.606,-178.098,5.583,148.408
C07244=1232.789,127.785,-49.587,-178.101,5.583,148.409
C07245=1232.793,127.537,-49.566,-178.103,5.582,148.409
C07246=1232.798,127.287,-49.547,-178.106,5.581,148.410
C07247=1232.803,127.039,-49.527,-178.109,5.580,148.411
C07248=1232.808,126.789,-49.506,-178.111,5.579,148.411
C07249=1232.813,126.540,-49.486,-178.114,5.578,148.412
C07250=1232.818,126.291,-49.466,-178.116,5.577,148.412
C07251=1232.822,126.041,-49.446,-178.119,5.575,148.413
C07252=1232.827,125.792,-49.425,-178.121,5.574,148.413
C07253=1232.832,125.544,-49.406,-178.124,5.574,148.414
C07254=1232.837,125.295,-49.386,-178.126,5.573,148.414
C07255=1232.841,125.045,-49.366,-178.129,5.571,148.415
C07256=1232.846,124.796,-49.346,-178.132,5.571,148.415
C07257=1232.850,124.547,-49.326,-178.134,5.570,148.416
C07258=1232.856,124.297,-49.305,-178.137,5.568,148.416
C07259=1232.861,124.048,-49.286,-178.139,5.568,148.417
C07260=1232.865,123.799,-49.266,-178.142,5.567,148.417
C07261=1232.870,123.550,-49.246,-178.144,5.566,148.418
C07262=1232.875,123.301,-49.225,-178.147,5.564,148.419
C07263=1232.879,123.051,-49.206,-178.149,5.564,148.419
C07264=1232.884,122.803,-49.186,-178.152,5.563,148.420
C07265=1232.889,122.554,-49.166,-178.154,5.562,148.420
C07266=1232.894,122.305,-49.146,-178.157,5.561,148.421
C07267=1232.898,122.055,-49.126,-178.159,5.560,148.421
C07268=1232.904,121.806,-49.107,-178.162,5.559,148.422
C07269=1232.908,121.557,-49.086,-178.164,5.558,148.422
C07270=1232.913,121.308,-49.067,-178.167,5.556,148.423
C07271=1232.918,121.058,-49.047,-178.170,5.556,148.424
C07272=1232.923,120.810,-49.027,-178.172,5.555,148.424
C07273=1232.927,120.560,-49.008,-178.175,5.554,148.425
C07274=1232.932,120.311,-48.988,-178.177,5.554,148.425
C07275=1232.937,120.062,-48.967,-178.180,5.552,148.426
C07276=1232.942,119.813,-48.948,-178.183,5.551,148.426
C07277=1232.947,119.563,-48.929,-178.185,5.550,148.427
C07278=1232.951,119.314,-48.908,-178.187,5.550,148.427
C07279=1232.956,119.065,-48.889,-178.190,5.548,148.428
C07280=1232.961,118.816,-48.869,-178.193,5.547,148.428
C07281=1232.966,118.567,-48.849,-178.195,5.547,148.429
C07282=1232.970,118.318,-48.830,-178.197,5.546,148.429
C07283=1232.975,118.069,-48.810,-178.200,5.544,148.430
C07284=1232.980,117.819,-48.791,-178.203,5.543,148.431
C07285=1232.984,117.570,-48.770,-178.205,5.542,148.431
C07286=1232.989,117.321,-48.751,-178.208,5.542,148.432
C07287=1232.994,117.072,-48.732,-178.210,5.541,148.432
C07288=1232.999,116.822,-48.712,-178.213,5.539,148.433
C07289=1233.003,116.573,-48.691,-178.216,5.539,148.433
C07290=1233.009,116.325,-48.672,-178.218,5.538,148.434
C07291=1233.013,116.075,-48.653,-178.220,5.537,148.434
C07292=1233.017,115.826,-48.633,-178.223,5.537,148.435
C07293=1233.023,115.577,-48.614,-178.226,5.535,148.435
C07294=1233.028,115.327,-48.595,-178.228,5.534,148.436
